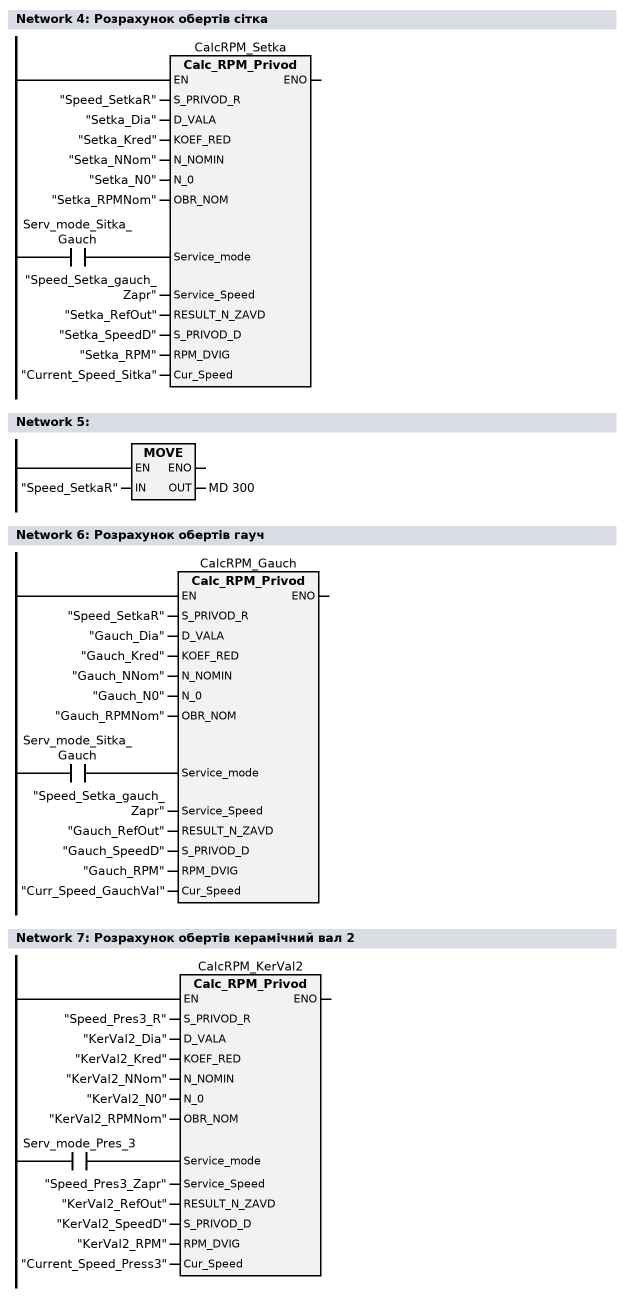
NETWORK
TITLE = Розрахунок обертів сітка
      A     "Serv_mode_Sitka_Gauch";
      =     L 0.0;
      BLD   103;
      CALL  "Calc_RPM_Privod" , "CalcRPM_Setka" (
           S_PRIVOD_R               := "Speed_SetkaR",
           D_VALA                   := "Setka_Dia",
           KOEF_RED                 := "Setka_Kred",
           N_NOMIN                  := "Setka_NNom",
           N_0                      := "Setka_N0",
           OBR_NOM                  := "Setka_RPMNom",
           Service_mode             := L 0.0,
           Service_Speed            := "Speed_Setka_gauch_Zapr",
           RESULT_N_ZAVD            := "Setka_RefOut",
           S_PRIVOD_D               := "Setka_SpeedD",
           RPM_DVIG                 := "Setka_RPM",
           Cur_Speed                := "Current_Speed_Sitka");
      NOP   0;
NETWORK
TITLE =
      L     "Speed_SetkaR";
      T     MD 300;
      NOP   0;
NETWORK
TITLE = Розрахунок обертів гауч
      A     "Serv_mode_Sitka_Gauch";
      =     L 0.0;
      BLD   103;
      CALL  "Calc_RPM_Privod" , "CalcRPM_Gauch" (
           S_PRIVOD_R               := "Speed_SetkaR",
           D_VALA                   := "Gauch_Dia",
           KOEF_RED                 := "Gauch_Kred",
           N_NOMIN                  := "Gauch_NNom",
           N_0                      := "Gauch_N0",
           OBR_NOM                  := "Gauch_RPMNom",
           Service_mode             := L 0.0,
           Service_Speed            := "Speed_Setka_gauch_Zapr",
           RESULT_N_ZAVD            := "Gauch_RefOut",
           S_PRIVOD_D               := "Gauch_SpeedD",
           RPM_DVIG                 := "Gauch_RPM",
           Cur_Speed                := "Curr_Speed_GauchVal");
      NOP   0;
NETWORK
TITLE = Розрахунок обертів керамічний вал 2
      A     "Serv_mode_Pres_3";
      =     L 0.0;
      BLD   103;
      CALL  "Calc_RPM_Privod" , "CalcRPM_KerVal2" (
           S_PRIVOD_R               := "Speed_Pres3_R",
           D_VALA                   := "KerVal2_Dia",
           KOEF_RED                 := "KerVal2_Kred",
           N_NOMIN                  := "KerVal2_NNom",
           N_0                      := "KerVal2_N0",
           OBR_NOM                  := "KerVal2_RPMNom",
           Service_mode             := L 0.0,
           Service_Speed            := "Speed_Pres3_Zapr",
           RESULT_N_ZAVD            := "KerVal2_RefOut",
           S_PRIVOD_D               := "KerVal2_SpeedD",
           RPM_DVIG                 := "KerVal2_RPM",
           Cur_Speed                := "Current_Speed_Press3");
      NOP   0;
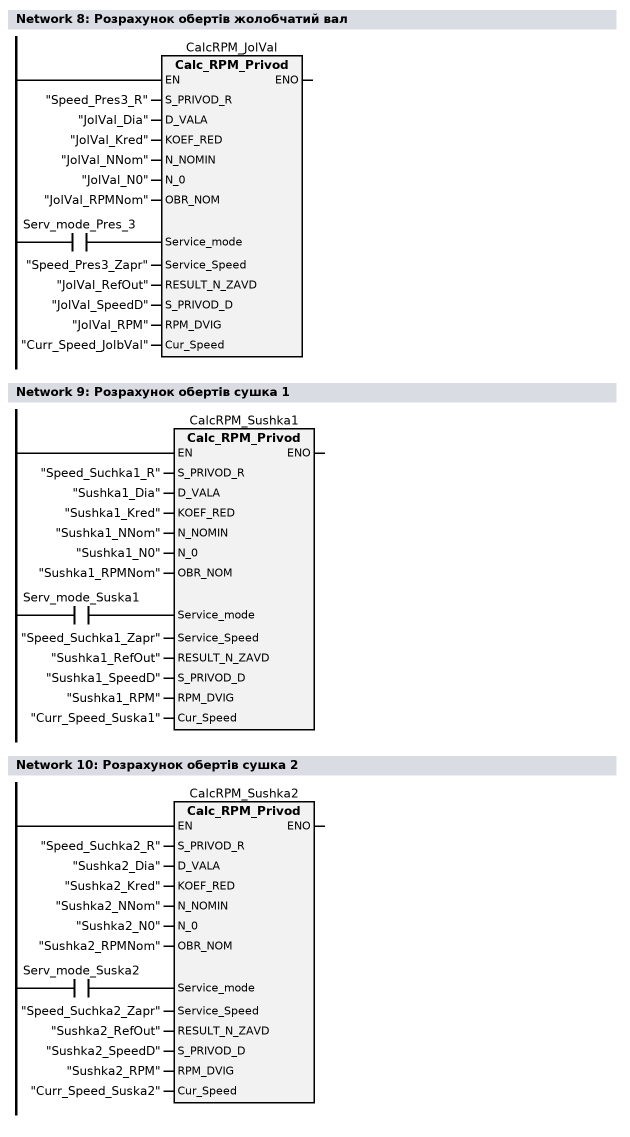
NETWORK
TITLE = Розрахунок обертів жолобчатий вал
      A     "Serv_mode_Pres_3";
      =     L 0.0;
      BLD   103;
      CALL  "Calc_RPM_Privod" , "CalcRPM_JolVal" (
           S_PRIVOD_R               := "Speed_Pres3_R",
           D_VALA                   := "JolVal_Dia",
           KOEF_RED                 := "JolVal_Kred",
           N_NOMIN                  := "JolVal_NNom",
           N_0                      := "JolVal_N0",
           OBR_NOM                  := "JolVal_RPMNom",
           Service_mode             := L 0.0,
           Service_Speed            := "Speed_Pres3_Zapr",
           RESULT_N_ZAVD            := "JolVal_RefOut",
           S_PRIVOD_D               := "JolVal_SpeedD",
           RPM_DVIG                 := "JolVal_RPM",
           Cur_Speed                := "Curr_Speed_JolbVal");
      NOP   0;
NETWORK
TITLE = Розрахунок обертів сушка 1
      A     "Serv_mode_Suska1";
      =     L 0.0;
      BLD   103;
      CALL  "Calc_RPM_Privod" , "CalcRPM_Sushka1" (
           S_PRIVOD_R               := "Speed_Suchka1_R",
           D_VALA                   := "Sushka1_Dia",
           KOEF_RED                 := "Sushka1_Kred",
           N_NOMIN                  := "Sushka1_NNom",
           N_0                      := "Sushka1_N0",
           OBR_NOM                  := "Sushka1_RPMNom",
           Service_mode             := L 0.0,
           Service_Speed            := "Speed_Suchka1_Zapr",
           RESULT_N_ZAVD            := "Sushka1_RefOut",
           S_PRIVOD_D               := "Sushka1_SpeedD",
           RPM_DVIG                 := "Sushka1_RPM",
           Cur_Speed                := "Curr_Speed_Suska1");
      NOP   0;
NETWORK
TITLE = Розрахунок обертів сушка 2
      A     "Serv_mode_Suska2";
      =     L 0.0;
      BLD   103;
      CALL  "Calc_RPM_Privod" , "CalcRPM_Sushka2" (
           S_PRIVOD_R               := "Speed_Suchka2_R",
           D_VALA                   := "Sushka2_Dia",
           KOEF_RED                 := "Sushka2_Kred",
           N_NOMIN                  := "Sushka2_NNom",
           N_0                      := "Sushka2_N0",
           OBR_NOM                  := "Sushka2_RPMNom",
           Service_mode             := L 0.0,
           Service_Speed            := "Speed_Suchka2_Zapr",
           RESULT_N_ZAVD            := "Sushka2_RefOut",
           S_PRIVOD_D               := "Sushka2_SpeedD",
           RPM_DVIG                 := "Sushka2_RPM",
           Cur_Speed                := "Curr_Speed_Suska2");
      NOP   0;
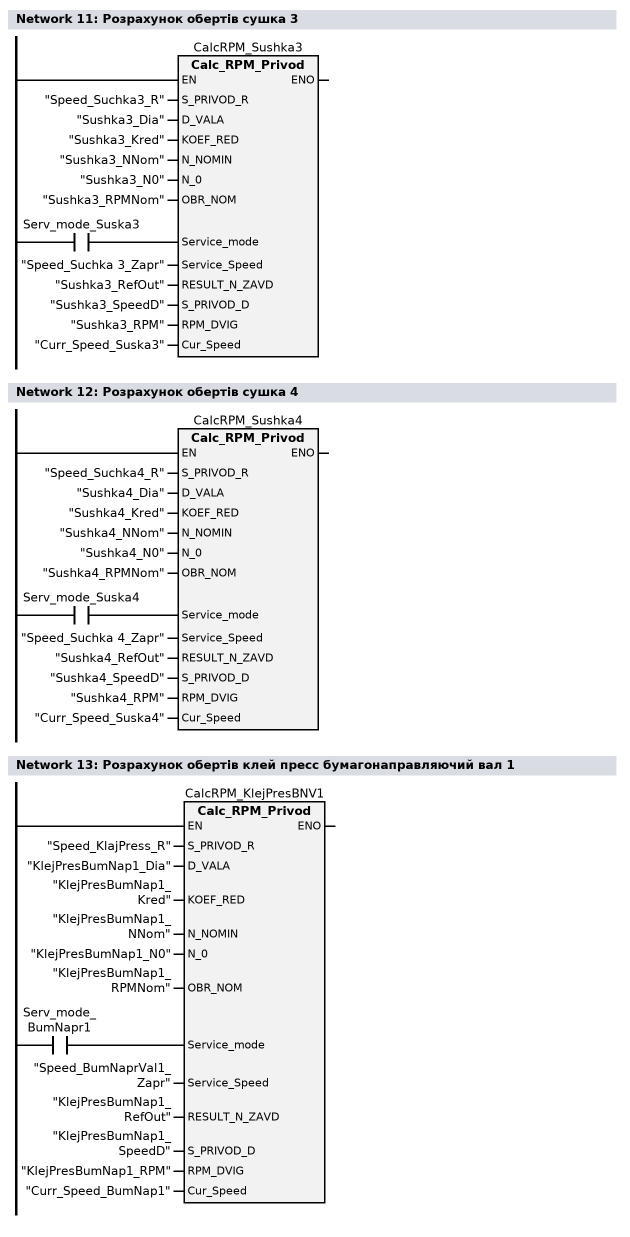
NETWORK
TITLE = Розрахунок обертів сушка 3
      A     "Serv_mode_Suska3";
      =     L 0.0;
      BLD   103;
      CALL  "Calc_RPM_Privod" , "CalcRPM_Sushka3" (
           S_PRIVOD_R               := "Speed_Suchka3_R",
           D_VALA                   := "Sushka3_Dia",
           KOEF_RED                 := "Sushka3_Kred",
           N_NOMIN                  := "Sushka3_NNom",
           N_0                      := "Sushka3_N0",
           OBR_NOM                  := "Sushka3_RPMNom",
           Service_mode             := L 0.0,
           Service_Speed            := "Speed_Suchka 3_Zapr",
           RESULT_N_ZAVD            := "Sushka3_RefOut",
           S_PRIVOD_D               := "Sushka3_SpeedD",
           RPM_DVIG                 := "Sushka3_RPM",
           Cur_Speed                := "Curr_Speed_Suska3");
      NOP   0;
NETWORK
TITLE = Розрахунок обертів сушка 4
      A     "Serv_mode_Suska4";
      =     L 0.0;
      BLD   103;
      CALL  "Calc_RPM_Privod" , "CalcRPM_Sushka4" (
           S_PRIVOD_R               := "Speed_Suchka4_R",
           D_VALA                   := "Sushka4_Dia",
           KOEF_RED                 := "Sushka4_Kred",
           N_NOMIN                  := "Sushka4_NNom",
           N_0                      := "Sushka4_N0",
           OBR_NOM                  := "Sushka4_RPMNom",
           Service_mode             := L 0.0,
           Service_Speed            := "Speed_Suchka 4_Zapr",
           RESULT_N_ZAVD            := "Sushka4_RefOut",
           S_PRIVOD_D               := "Sushka4_SpeedD",
           RPM_DVIG                 := "Sushka4_RPM",
           Cur_Speed                := "Curr_Speed_Suska4");
      NOP   0;
NETWORK
TITLE = Розрахунок обертів клей пресс бумагонаправляючий вал 1
      A     "Serv_mode_BumNapr1";
      =     L 0.0;
      BLD   103;
      CALL  "Calc_RPM_Privod" , "CalcRPM_KlejPresBNV1" (
           S_PRIVOD_R               := "Speed_KlajPress_R",
           D_VALA                   := "KlejPresBumNap1_Dia",
           KOEF_RED                 := "KlejPresBumNap1_Kred",
           N_NOMIN                  := "KlejPresBumNap1_NNom",
           N_0                      := "KlejPresBumNap1_N0",
           OBR_NOM                  := "KlejPresBumNap1_RPMNom",
           Service_mode             := L 0.0,
           Service_Speed            := "Speed_BumNaprVal1_Zapr",
           RESULT_N_ZAVD            := "KlejPresBumNap1_RefOut",
           S_PRIVOD_D               := "KlejPresBumNap1_SpeedD",
           RPM_DVIG                 := "KlejPresBumNap1_RPM",
           Cur_Speed                := "Curr_Speed_BumNap1");
      NOP   0;
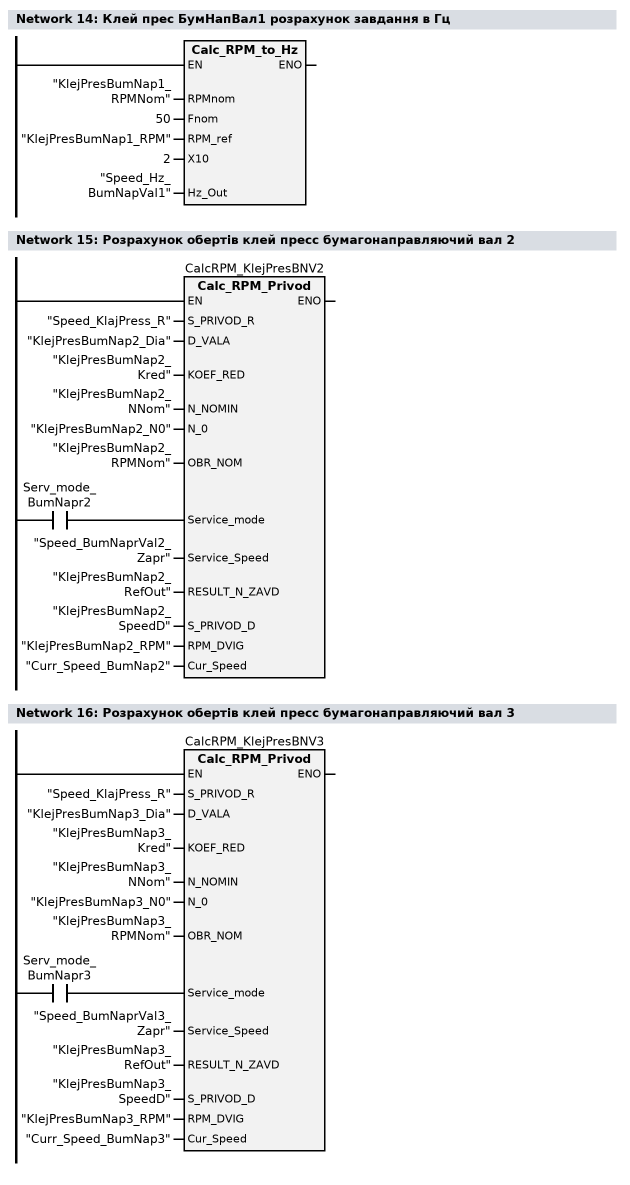
NETWORK
TITLE = Клей прес БумНапВал1 розрахунок завдання в Гц
      CALL  "Calc_RPM_to_Hz" (
           RPMnom                   := "KlejPresBumNap1_RPMNom",
           Fnom                     := 50,
           RPM_ref                  := "KlejPresBumNap1_RPM",
           X10                      := 2,
           Hz_Out                   := "Speed_Hz_BumNapVal1");
      NOP   0;
NETWORK
TITLE = Розрахунок обертів клей пресс бумагонаправляючий вал 2
      A     "Serv_mode_BumNapr2";
      =     L 0.0;
      BLD   103;
      CALL  "Calc_RPM_Privod" , "CalcRPM_KlejPresBNV2" (
           S_PRIVOD_R               := "Speed_KlajPress_R",
           D_VALA                   := "KlejPresBumNap2_Dia",
           KOEF_RED                 := "KlejPresBumNap2_Kred",
           N_NOMIN                  := "KlejPresBumNap2_NNom",
           N_0                      := "KlejPresBumNap2_N0",
           OBR_NOM                  := "KlejPresBumNap2_RPMNom",
           Service_mode             := L 0.0,
           Service_Speed            := "Speed_BumNaprVal2_Zapr",
           RESULT_N_ZAVD            := "KlejPresBumNap2_RefOut",
           S_PRIVOD_D               := "KlejPresBumNap2_SpeedD",
           RPM_DVIG                 := "KlejPresBumNap2_RPM",
           Cur_Speed                := "Curr_Speed_BumNap2");
      NOP   0;
NETWORK
TITLE = Розрахунок обертів клей пресс бумагонаправляючий вал 3
      A     "Serv_mode_BumNapr3";
      =     L 0.0;
      BLD   103;
      CALL  "Calc_RPM_Privod" , "CalcRPM_KlejPresBNV3" (
           S_PRIVOD_R               := "Speed_KlajPress_R",
           D_VALA                   := "KlejPresBumNap3_Dia",
           KOEF_RED                 := "KlejPresBumNap3_Kred",
           N_NOMIN                  := "KlejPresBumNap3_NNom",
           N_0                      := "KlejPresBumNap3_N0",
           OBR_NOM                  := "KlejPresBumNap3_RPMNom",
           Service_mode             := L 0.0,
           Service_Speed            := "Speed_BumNaprVal3_Zapr",
           RESULT_N_ZAVD            := "KlejPresBumNap3_RefOut",
           S_PRIVOD_D               := "KlejPresBumNap3_SpeedD",
           RPM_DVIG                 := "KlejPresBumNap3_RPM",
           Cur_Speed                := "Curr_Speed_BumNap3");
      NOP   0;
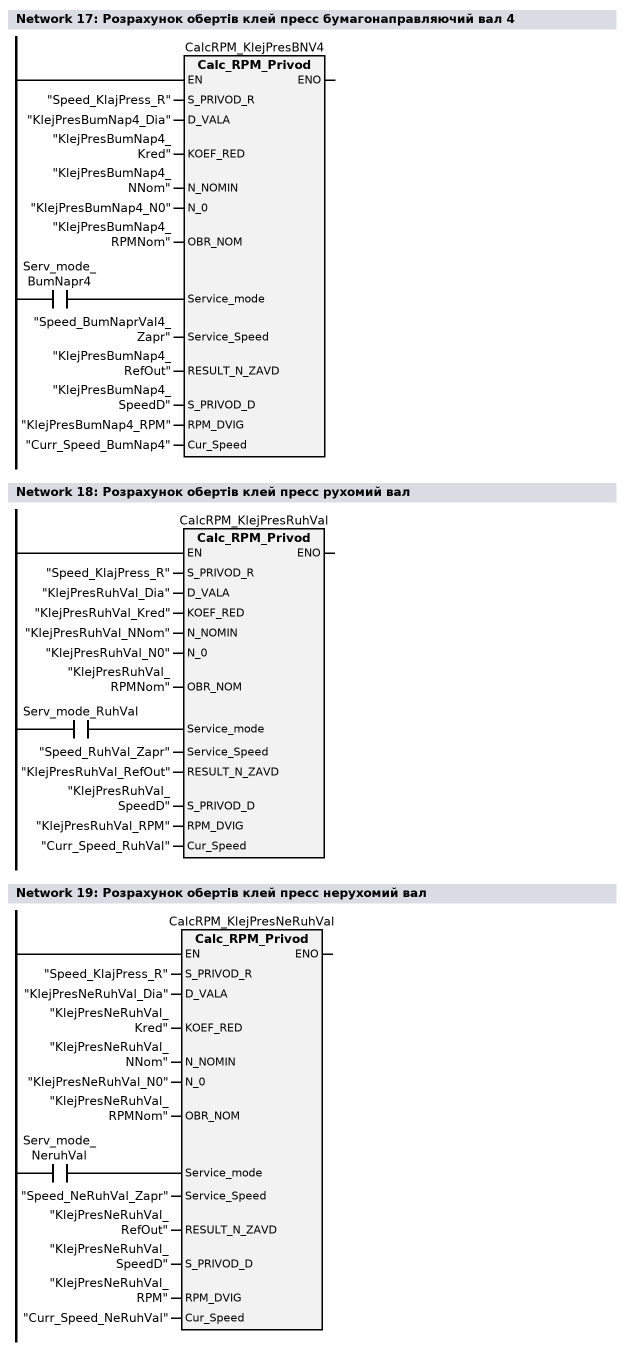
NETWORK
TITLE = Розрахунок обертів клей пресс бумагонаправляючий вал 4
      A     "Serv_mode_BumNapr4";
      =     L 0.0;
      BLD   103;
      CALL  "Calc_RPM_Privod" , "CalcRPM_KlejPresBNV4" (
           S_PRIVOD_R               := "Speed_KlajPress_R",
           D_VALA                   := "KlejPresBumNap4_Dia",
           KOEF_RED                 := "KlejPresBumNap4_Kred",
           N_NOMIN                  := "KlejPresBumNap4_NNom",
           N_0                      := "KlejPresBumNap4_N0",
           OBR_NOM                  := "KlejPresBumNap4_RPMNom",
           Service_mode             := L 0.0,
           Service_Speed            := "Speed_BumNaprVal4_Zapr",
           RESULT_N_ZAVD            := "KlejPresBumNap4_RefOut",
           S_PRIVOD_D               := "KlejPresBumNap4_SpeedD",
           RPM_DVIG                 := "KlejPresBumNap4_RPM",
           Cur_Speed                := "Curr_Speed_BumNap4");
      NOP   0;
NETWORK
TITLE = Розрахунок обертів клей пресс рухомий вал
      A     "Serv_mode_RuhVal";
      =     L 0.0;
      BLD   103;
      CALL  "Calc_RPM_Privod" , "CalcRPM_KlejPresRuhVal" (
           S_PRIVOD_R               := "Speed_KlajPress_R",
           D_VALA                   := "KlejPresRuhVal_Dia",
           KOEF_RED                 := "KlejPresRuhVal_Kred",
           N_NOMIN                  := "KlejPresRuhVal_NNom",
           N_0                      := "KlejPresRuhVal_N0",
           OBR_NOM                  := "KlejPresRuhVal_RPMNom",
           Service_mode             := L 0.0,
           Service_Speed            := "Speed_RuhVal_Zapr",
           RESULT_N_ZAVD            := "KlejPresRuhVal_RefOut",
           S_PRIVOD_D               := "KlejPresRuhVal_SpeedD",
           RPM_DVIG                 := "KlejPresRuhVal_RPM",
           Cur_Speed                := "Curr_Speed_RuhVal");
      NOP   0;
NETWORK
TITLE = Розрахунок обертів клей пресс нерухомий вал
      A     "Serv_mode_NeruhVal";
      =     L 0.0;
      BLD   103;
      CALL  "Calc_RPM_Privod" , "CalcRPM_KlejPresNeRuhVal" (
           S_PRIVOD_R               := "Speed_KlajPress_R",
           D_VALA                   := "KlejPresNeRuhVal_Dia",
           KOEF_RED                 := "KlejPresNeRuhVal_Kred",
           N_NOMIN                  := "KlejPresNeRuhVal_NNom",
           N_0                      := "KlejPresNeRuhVal_N0",
           OBR_NOM                  := "KlejPresNeRuhVal_RPMNom",
           Service_mode             := L 0.0,
           Service_Speed            := "Speed_NeRuhVal_Zapr",
           RESULT_N_ZAVD            := "KlejPresNeRuhVal_RefOut",
           S_PRIVOD_D               := "KlejPresNeRuhVal_SpeedD",
           RPM_DVIG                 := "KlejPresNeRuhVal_RPM",
           Cur_Speed                := "Curr_Speed_NeRuhVal");
      NOP   0;
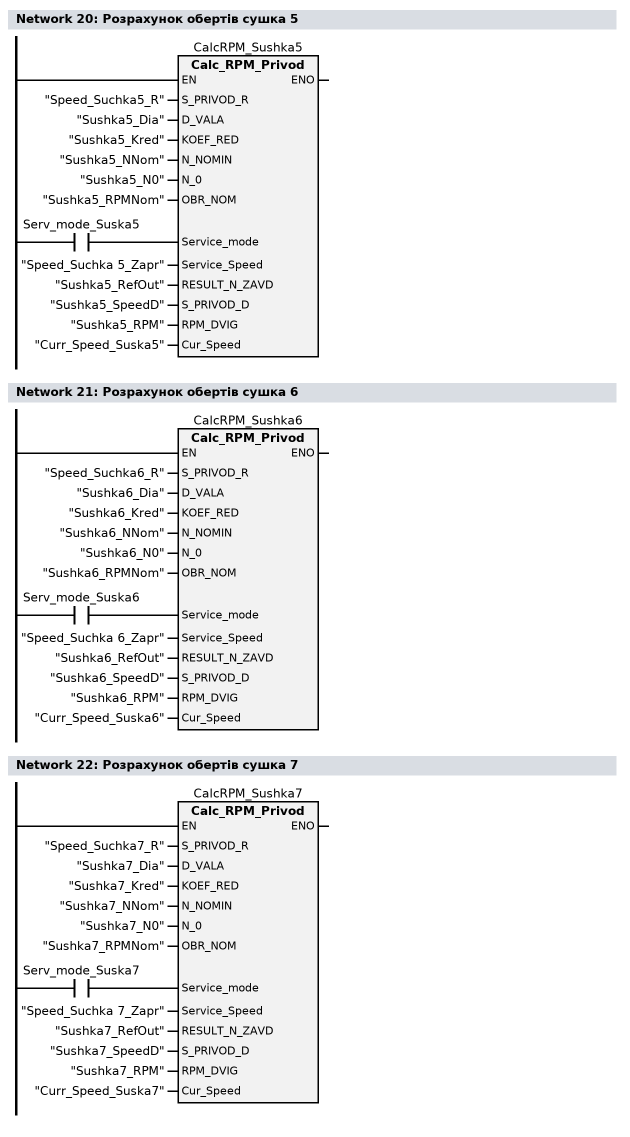
NETWORK
TITLE = Розрахунок обертів сушка 5
      A     "Serv_mode_Suska5";
      =     L 0.0;
      BLD   103;
      CALL  "Calc_RPM_Privod" , "CalcRPM_Sushka5" (
           S_PRIVOD_R               := "Speed_Suchka5_R",
           D_VALA                   := "Sushka5_Dia",
           KOEF_RED                 := "Sushka5_Kred",
           N_NOMIN                  := "Sushka5_NNom",
           N_0                      := "Sushka5_N0",
           OBR_NOM                  := "Sushka5_RPMNom",
           Service_mode             := L 0.0,
           Service_Speed            := "Speed_Suchka 5_Zapr",
           RESULT_N_ZAVD            := "Sushka5_RefOut",
           S_PRIVOD_D               := "Sushka5_SpeedD",
           RPM_DVIG                 := "Sushka5_RPM",
           Cur_Speed                := "Curr_Speed_Suska5");
      NOP   0;
NETWORK
TITLE = Розрахунок обертів сушка 6
      A     "Serv_mode_Suska6";
      =     L 0.0;
      BLD   103;
      CALL  "Calc_RPM_Privod" , "CalcRPM_Sushka6" (
           S_PRIVOD_R               := "Speed_Suchka6_R",
           D_VALA                   := "Sushka6_Dia",
           KOEF_RED                 := "Sushka6_Kred",
           N_NOMIN                  := "Sushka6_NNom",
           N_0                      := "Sushka6_N0",
           OBR_NOM                  := "Sushka6_RPMNom",
           Service_mode             := L 0.0,
           Service_Speed            := "Speed_Suchka 6_Zapr",
           RESULT_N_ZAVD            := "Sushka6_RefOut",
           S_PRIVOD_D               := "Sushka6_SpeedD",
           RPM_DVIG                 := "Sushka6_RPM",
           Cur_Speed                := "Curr_Speed_Suska6");
      NOP   0;
NETWORK
TITLE = Розрахунок обертів сушка 7
      A     "Serv_mode_Suska7";
      =     L 0.0;
      BLD   103;
      CALL  "Calc_RPM_Privod" , "CalcRPM_Sushka7" (
           S_PRIVOD_R               := "Speed_Suchka7_R",
           D_VALA                   := "Sushka7_Dia",
           KOEF_RED                 := "Sushka7_Kred",
           N_NOMIN                  := "Sushka7_NNom",
           N_0                      := "Sushka7_N0",
           OBR_NOM                  := "Sushka7_RPMNom",
           Service_mode             := L 0.0,
           Service_Speed            := "Speed_Suchka 7_Zapr",
           RESULT_N_ZAVD            := "Sushka7_RefOut",
           S_PRIVOD_D               := "Sushka7_SpeedD",
           RPM_DVIG                 := "Sushka7_RPM",
           Cur_Speed                := "Curr_Speed_Suska7");
      NOP   0;
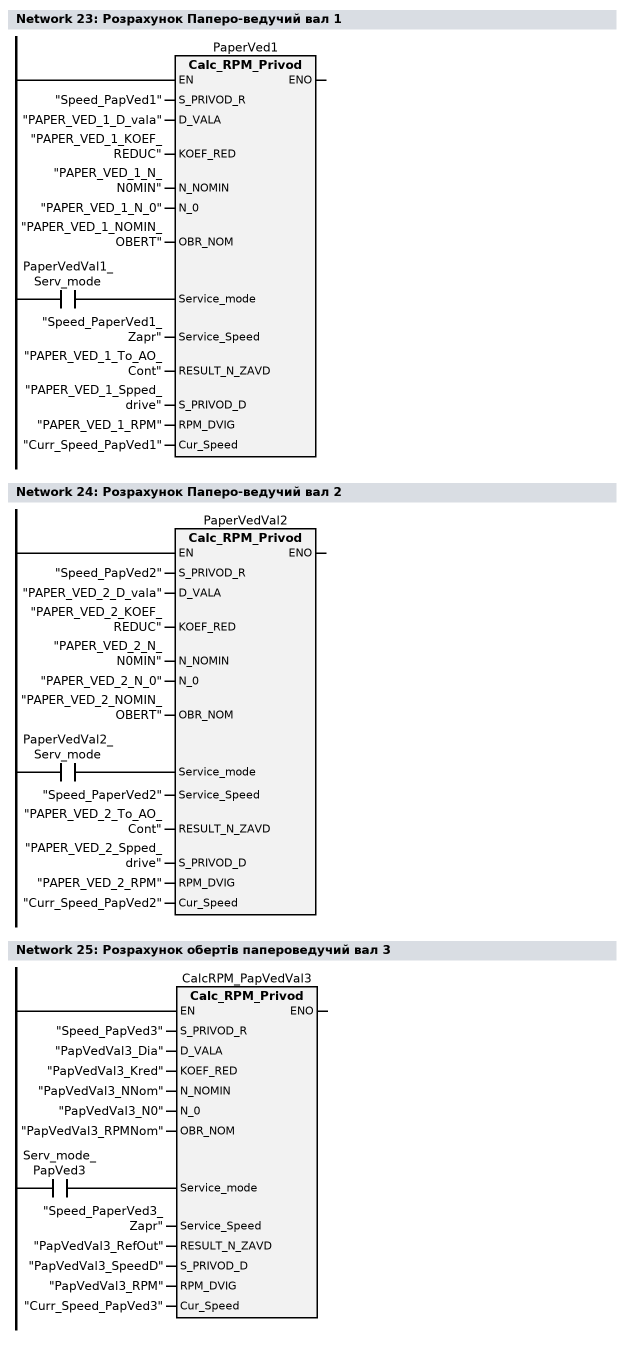
NETWORK
TITLE = Розрахунок Паперо-ведучий вал 1
//********************************************
//
      A     "PaperVedVal1_Serv_mode";
      =     L 0.0;
      BLD   103;
      CALL  "Calc_RPM_Privod" , "PaperVed1" (
           S_PRIVOD_R               := "Speed_PapVed1",
           D_VALA                   := "PAPER_VED_1_D_vala",
           KOEF_RED                 := "PAPER_VED_1_KOEF_REDUC",
           N_NOMIN                  := "PAPER_VED_1_N_N0MIN",
           N_0                      := "PAPER_VED_1_N_0",
           OBR_NOM                  := "PAPER_VED_1_NOMIN_OBERT",
           Service_mode             := L 0.0,
           Service_Speed            := "Speed_PaperVed1_Zapr",
           RESULT_N_ZAVD            := "PAPER_VED_1_To_AO_Cont",
           S_PRIVOD_D               := "PAPER_VED_1_Spped_drive",
           RPM_DVIG                 := "PAPER_VED_1_RPM",
           Cur_Speed                := "Curr_Speed_PapVed1");
      NOP   0;
NETWORK
TITLE = Розрахунок Паперо-ведучий вал 2
//*********************************************
//
      A     "PaperVedVal2_Serv_mode";
      =     L 0.0;
      BLD   103;
      CALL  "Calc_RPM_Privod" , "PaperVedVal2" (
           S_PRIVOD_R               := "Speed_PapVed2",
           D_VALA                   := "PAPER_VED_2_D_vala",
           KOEF_RED                 := "PAPER_VED_2_KOEF_REDUC",
           N_NOMIN                  := "PAPER_VED_2_N_N0MIN",
           N_0                      := "PAPER_VED_2_N_0",
           OBR_NOM                  := "PAPER_VED_2_NOMIN_OBERT",
           Service_mode             := L 0.0,
           Service_Speed            := "Speed_PaperVed2",
           RESULT_N_ZAVD            := "PAPER_VED_2_To_AO_Cont",
           S_PRIVOD_D               := "PAPER_VED_2_Spped_drive",
           RPM_DVIG                 := "PAPER_VED_2_RPM",
           Cur_Speed                := "Curr_Speed_PapVed2");
      NOP   0;
NETWORK
TITLE = Розрахунок обертів папероведучий вал 3
//****************************************************
//
      A     "Serv_mode_PapVed3";
      =     L 0.0;
      BLD   103;
      CALL  "Calc_RPM_Privod" , "CalcRPM_PapVedVal3" (
           S_PRIVOD_R               := "Speed_PapVed3",
           D_VALA                   := "PapVedVal3_Dia",
           KOEF_RED                 := "PapVedVal3_Kred",
           N_NOMIN                  := "PapVedVal3_NNom",
           N_0                      := "PapVedVal3_N0",
           OBR_NOM                  := "PapVedVal3_RPMNom",
           Service_mode             := L 0.0,
           Service_Speed            := "Speed_PaperVed3_Zapr",
           RESULT_N_ZAVD            := "PapVedVal3_RefOut",
           S_PRIVOD_D               := "PapVedVal3_SpeedD",
           RPM_DVIG                 := "PapVedVal3_RPM",
           Cur_Speed                := "Curr_Speed_PapVed3");
      NOP   0;
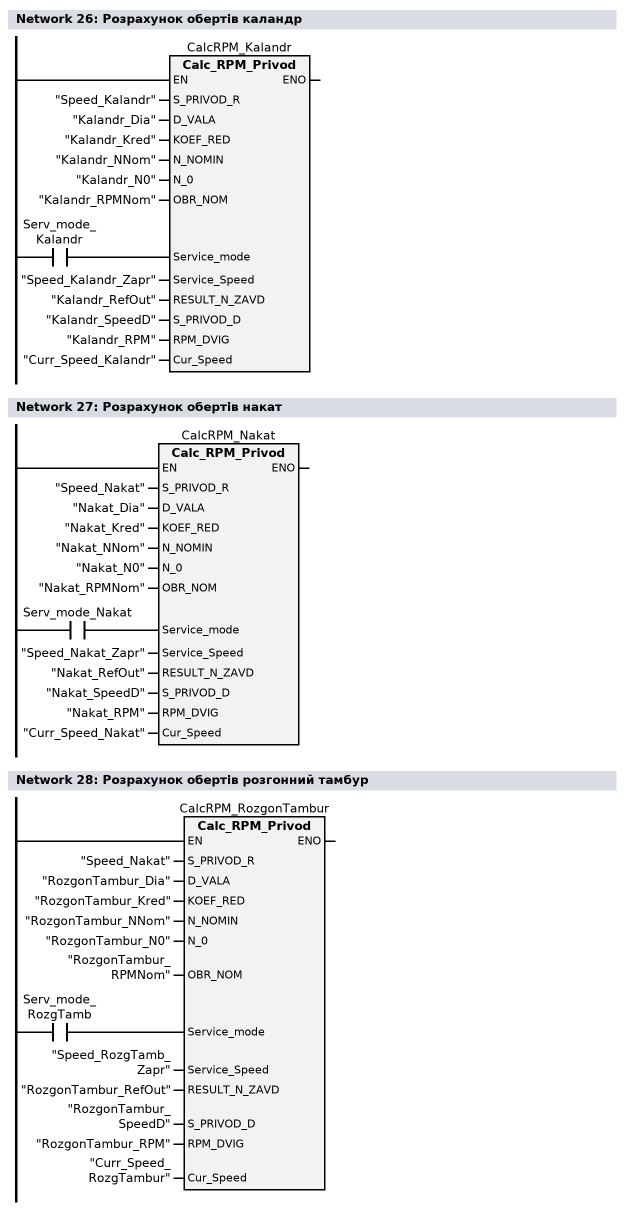
NETWORK
TITLE = Розрахунок обертів каландр
      A     "Serv_mode_Kalandr";
      =     L 0.0;
      BLD   103;
      CALL  "Calc_RPM_Privod" , "CalcRPM_Kalandr" (
           S_PRIVOD_R               := "Speed_Kalandr",
           D_VALA                   := "Kalandr_Dia",
           KOEF_RED                 := "Kalandr_Kred",
           N_NOMIN                  := "Kalandr_NNom",
           N_0                      := "Kalandr_N0",
           OBR_NOM                  := "Kalandr_RPMNom",
           Service_mode             := L 0.0,
           Service_Speed            := "Speed_Kalandr_Zapr",
           RESULT_N_ZAVD            := "Kalandr_RefOut",
           S_PRIVOD_D               := "Kalandr_SpeedD",
           RPM_DVIG                 := "Kalandr_RPM",
           Cur_Speed                := "Curr_Speed_Kalandr");
      NOP   0;
NETWORK
TITLE = Розрахунок обертів накат
      A     "Serv_mode_Nakat";
      =     L 0.0;
      BLD   103;
      CALL  "Calc_RPM_Privod" , "CalcRPM_Nakat" (
           S_PRIVOD_R               := "Speed_Nakat",
           D_VALA                   := "Nakat_Dia",
           KOEF_RED                 := "Nakat_Kred",
           N_NOMIN                  := "Nakat_NNom",
           N_0                      := "Nakat_N0",
           OBR_NOM                  := "Nakat_RPMNom",
           Service_mode             := L 0.0,
           Service_Speed            := "Speed_Nakat_Zapr",
           RESULT_N_ZAVD            := "Nakat_RefOut",
           S_PRIVOD_D               := "Nakat_SpeedD",
           RPM_DVIG                 := "Nakat_RPM",
           Cur_Speed                := "Curr_Speed_Nakat");
      NOP   0;
NETWORK
TITLE = Розрахунок обертів розгонний тамбур
      A     "Serv_mode_RozgTamb";
      =     L 0.0;
      BLD   103;
      CALL  "Calc_RPM_Privod" , "CalcRPM_RozgonTambur" (
           S_PRIVOD_R               := "Speed_Nakat",
           D_VALA                   := "RozgonTambur_Dia",
           KOEF_RED                 := "RozgonTambur_Kred",
           N_NOMIN                  := "RozgonTambur_NNom",
           N_0                      := "RozgonTambur_N0",
           OBR_NOM                  := "RozgonTambur_RPMNom",
           Service_mode             := L 0.0,
           Service_Speed            := "Speed_RozgTamb_Zapr",
           RESULT_N_ZAVD            := "RozgonTambur_RefOut",
           S_PRIVOD_D               := "RozgonTambur_SpeedD",
           RPM_DVIG                 := "RozgonTambur_RPM",
           Cur_Speed                := "Curr_Speed_RozgTambur");
      NOP   0;
END_FUNCTION

FUNCTION "Speed_Intens" : VOID	// FC 12
VERSION : 0.1
VAR_TEMP
  Speed_1R : REAL ;
END_VAR
BEGIN
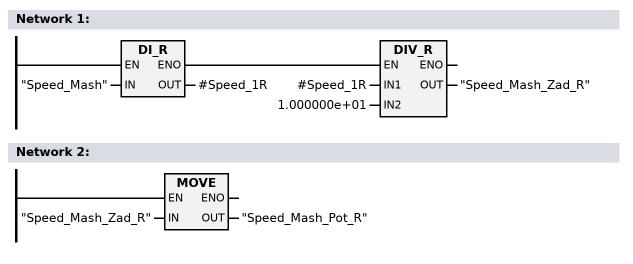
NETWORK
TITLE =
      A(;
      L     "Speed_Mash";
      DTR;
      T     #Speed_1R;
      SET;
      SAVE;
      CLR;
      A     BR;
      );
      JNB   _001;
      L     #Speed_1R;
      L     1.000000e+01;
      /R;
      T     "Speed_Mash_Zad_R";
_001: NOP   0;
NETWORK
TITLE =
      L     "Speed_Mash_Zad_R";
      T     "Speed_Mash_Pot_R";
      NOP   0;
END_FUNCTION

FUNCTION "Calc_RPM_to_Hz" : VOID	// FC 14
VERSION : 0.1
VAR_INPUT
  RPMnom : DINT ;
  Fnom : INT ;
  RPM_ref : DINT ;
  X10 : INT ;
END_VAR
VAR_OUTPUT
  Hz_Out : WORD ;
END_VAR
VAR_TEMP
  Fn_R : REAL ;
  Rn_R : REAL ;
  Rz_R : REAL ;
  Fnom_DI : DINT ;
  TEMP0 : REAL ;
  Fref_R : REAL ;
  TEMP10 : REAL ;
  TEMP1 : REAL ;
  Hz_Out_DI : DINT ;
END_VAR
BEGIN
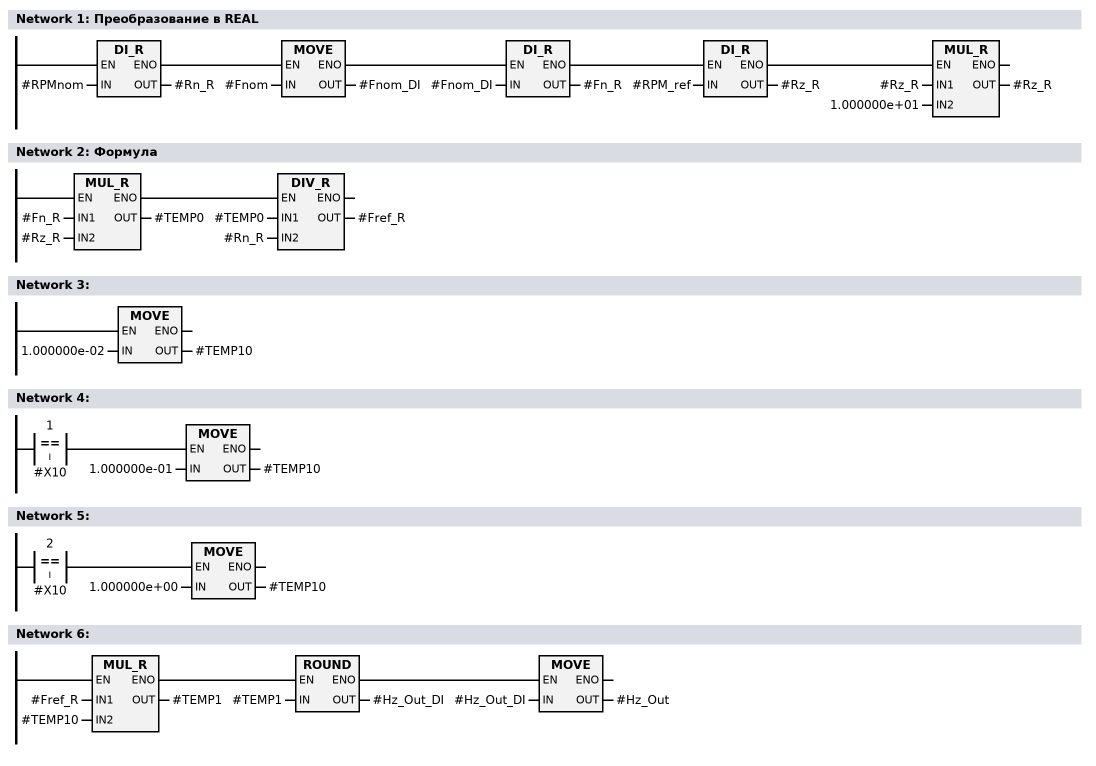
NETWORK
TITLE = Преобразование в REAL
      A(;
      A(;
      A(;
      A(;
      L     #RPMnom;
      DTR;
      T     #Rn_R;
      SET;
      SAVE;
      CLR;
      A     BR;
      );
      JNB   _001;
      L     #Fnom;
      T     #Fnom_DI;
      SET;
      SAVE;
      CLR;
_001: A     BR;
      );
      JNB   _002;
      L     #Fnom_DI;
      DTR;
      T     #Fn_R;
      SET;
      SAVE;
      CLR;
_002: A     BR;
      );
      JNB   _003;
      L     #RPM_ref;
      DTR;
      T     #Rz_R;
      SET;
      SAVE;
      CLR;
_003: A     BR;
      );
      JNB   _004;
      L     #Rz_R;
      L     1.000000e+01;
      *R;
      T     #Rz_R;
_004: NOP   0;
NETWORK
TITLE = Формула
      A(;
      L     #Fn_R;
      L     #Rz_R;
      *R;
      T     #TEMP0;
      AN    OV;
      SAVE;
      CLR;
      A     BR;
      );
      JNB   _005;
      L     #TEMP0;
      L     #Rn_R;
      /R;
      T     #Fref_R;
_005: NOP   0;
NETWORK
TITLE =
      L     1.000000e-02;
      T     #TEMP10;
      NOP   0;
NETWORK
TITLE =
      A(;
      L     1;
      L     #X10;
      ==I;
      );
      JNB   _006;
      L     1.000000e-01;
      T     #TEMP10;
_006: NOP   0;
NETWORK
TITLE =
      A(;
      L     2;
      L     #X10;
      ==I;
      );
      JNB   _007;
      L     1.000000e+00;
      T     #TEMP10;
_007: NOP   0;
NETWORK
TITLE =
      A(;
      A(;
      L     #Fref_R;
      L     #TEMP10;
      *R;
      T     #TEMP1;
      AN    OV;
      SAVE;
      CLR;
      A     BR;
      );
      JNB   _008;
      L     #TEMP1;
      RND;
      T     #Hz_Out_DI;
      AN    OV;
      SAVE;
      CLR;
_008: A     BR;
      );
      JNB   _009;
      L     #Hz_Out_DI;
      T     #Hz_Out;
_009: NOP   0;
END_FUNCTION

FUNCTION "Check_AlarmPPS" : VOID	// FC 30
VERSION : 0.1
VAR_INPUT
  Key_FU : BOOL ;
  Key_DozvilRun : BOOL ;
  Blokuvannja : BOOL ;
  AlarmPryvid : BOOL ;
  Warnunug_T : BOOL ;
  Alarm_T : BOOL ;
END_VAR
VAR_OUTPUT
  Cod_Err : WORD ;
  Privod_OK : BOOL ;
END_VAR
VAR_TEMP
  TEMP : BOOL ;
END_VAR
BEGIN
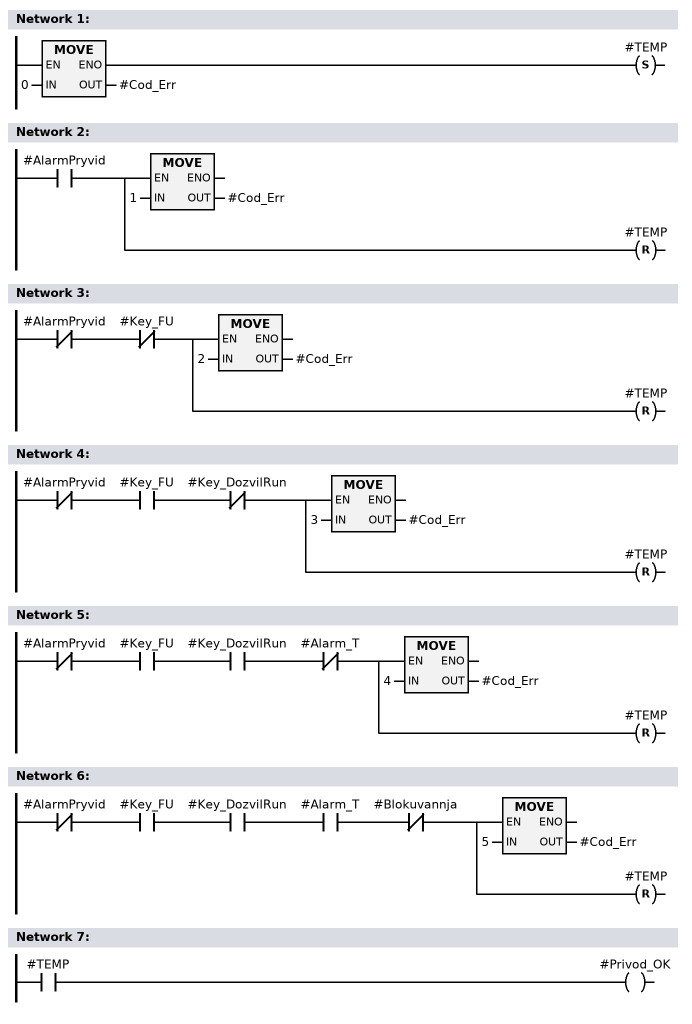
NETWORK
TITLE =
      L     0;
      T     #Cod_Err;
      SET;
      SAVE;
      CLR;
      A     BR;
      S     #TEMP;
NETWORK
TITLE =
      A     #AlarmPryvid;
      =     L 1.0;
      A     L 1.0;
      JNB   _001;
      L     1;
      T     #Cod_Err;
_001: NOP   0;
      A     L 1.0;
      BLD   102;
      R     #TEMP;
NETWORK
TITLE =
      AN    #AlarmPryvid;
      AN    #Key_FU;
      =     L 1.0;
      A     L 1.0;
      JNB   _002;
      L     2;
      T     #Cod_Err;
_002: NOP   0;
      A     L 1.0;
      BLD   102;
      R     #TEMP;
NETWORK
TITLE =
      AN    #AlarmPryvid;
      A     #Key_FU;
      AN    #Key_DozvilRun;
      =     L 1.0;
      A     L 1.0;
      JNB   _003;
      L     3;
      T     #Cod_Err;
_003: NOP   0;
      A     L 1.0;
      BLD   102;
      R     #TEMP;
NETWORK
TITLE =
      AN    #AlarmPryvid;
      A     #Key_FU;
      A     #Key_DozvilRun;
      AN    #Alarm_T;
      =     L 1.0;
      A     L 1.0;
      JNB   _004;
      L     4;
      T     #Cod_Err;
_004: NOP   0;
      A     L 1.0;
      BLD   102;
      R     #TEMP;
NETWORK
TITLE =
      AN    #AlarmPryvid;
      A     #Key_FU;
      A     #Key_DozvilRun;
      A     #Alarm_T;
      AN    #Blokuvannja;
      =     L 1.0;
      A     L 1.0;
      JNB   _005;
      L     5;
      T     #Cod_Err;
_005: NOP   0;
      A     L 1.0;
      BLD   102;
      R     #TEMP;
NETWORK
TITLE =
      A     #TEMP;
      =     #Privod_OK;
END_FUNCTION

// FC 216: know-how protected block, not included

DATA_BLOCK DB 60
VERSION : 0.0
"SEND"
BEGIN
END_DATA_BLOCK

DATA_BLOCK DB 61
VERSION : 0.0
"RECEIVE"
BEGIN
END_DATA_BLOCK

DATA_BLOCK "RS485_chenal1"	// DB 71
AUTHOR : VIPA
FAMILY : MODBUS
VERSION : 0.0
"RTU_MB_MASTER"
BEGIN
END_DATA_BLOCK

DATA_BLOCK "RS485_chanel2"	// DB 72
AUTHOR : VIPA
FAMILY : MODBUS
VERSION : 0.1
"RTU_MB_MASTER"
BEGIN
END_DATA_BLOCK

DATA_BLOCK "RS485_chanel3"	// DB 73
AUTHOR : VIPA
FAMILY : MODBUS
VERSION : 0.0
"RTU_MB_MASTER"
BEGIN
END_DATA_BLOCK

DATA_BLOCK "RS485_chanel4"	// DB 74
AUTHOR : VIPA
FAMILY : MODBUS
VERSION : 0.0
"RTU_MB_MASTER"
BEGIN
END_DATA_BLOCK

DATA_BLOCK "KerVal1"	// DB 101
VERSION : 0.1
"Calc_RPM_Privod"
BEGIN
END_DATA_BLOCK

DATA_BLOCK "ValGluchPerf"	// DB 102
VERSION : 0.0
"Calc_RPM_Privod"
BEGIN
END_DATA_BLOCK

DATA_BLOCK "VidsmokVal"	// DB 103
VERSION : 0.0
"Calc_RPM_Privod"
BEGIN
END_DATA_BLOCK

DATA_BLOCK "CalcRPM_Setka"	// DB 104
VERSION : 0.0
"Calc_RPM_Privod"
BEGIN
END_DATA_BLOCK

DATA_BLOCK "CalcRPM_Gauch"	// DB 105
VERSION : 0.0
"Calc_RPM_Privod"
BEGIN
END_DATA_BLOCK

DATA_BLOCK "CalcRPM_KerVal2"	// DB 106
VERSION : 0.0
"Calc_RPM_Privod"
BEGIN
END_DATA_BLOCK

DATA_BLOCK "CalcRPM_JolVal"	// DB 107
VERSION : 0.0
"Calc_RPM_Privod"
BEGIN
END_DATA_BLOCK

DATA_BLOCK "CalcRPM_Sushka1"	// DB 108
VERSION : 0.0
"Calc_RPM_Privod"
BEGIN
END_DATA_BLOCK

DATA_BLOCK "CalcRPM_Sushka2"	// DB 109
VERSION : 0.0
"Calc_RPM_Privod"
BEGIN
END_DATA_BLOCK

DATA_BLOCK "CalcRPM_Sushka3"	// DB 110
VERSION : 0.0
"Calc_RPM_Privod"
BEGIN
END_DATA_BLOCK

DATA_BLOCK "CalcRPM_Sushka4"	// DB 111
VERSION : 0.0
"Calc_RPM_Privod"
BEGIN
END_DATA_BLOCK

DATA_BLOCK "CalcRPM_KlejPresBNV1"	// DB 112
VERSION : 0.0
"Calc_RPM_Privod"
BEGIN
END_DATA_BLOCK

DATA_BLOCK "CalcRPM_KlejPresBNV2"	// DB 113
VERSION : 0.0
"Calc_RPM_Privod"
BEGIN
END_DATA_BLOCK

DATA_BLOCK "CalcRPM_KlejPresBNV3"	// DB 114
VERSION : 0.0
"Calc_RPM_Privod"
BEGIN
END_DATA_BLOCK

DATA_BLOCK "CalcRPM_KlejPresBNV4"	// DB 115
VERSION : 0.0
"Calc_RPM_Privod"
BEGIN
END_DATA_BLOCK

DATA_BLOCK "CalcRPM_KlejPresRuhVal"	// DB 116
VERSION : 0.0
"Calc_RPM_Privod"
BEGIN
END_DATA_BLOCK

DATA_BLOCK "CalcRPM_KlejPresNeRuhVal"	// DB 117
VERSION : 0.0
"Calc_RPM_Privod"
BEGIN
END_DATA_BLOCK

DATA_BLOCK "CalcRPM_Sushka5"	// DB 118
VERSION : 0.0
"Calc_RPM_Privod"
BEGIN
END_DATA_BLOCK

DATA_BLOCK "CalcRPM_Sushka6"	// DB 119
VERSION : 0.0
"Calc_RPM_Privod"
BEGIN
END_DATA_BLOCK

DATA_BLOCK "CalcRPM_Sushka7"	// DB 120
VERSION : 0.0
"Calc_RPM_Privod"
BEGIN
END_DATA_BLOCK

DATA_BLOCK "CalcRPM_Kalandr"	// DB 121
VERSION : 0.0
"Calc_RPM_Privod"
BEGIN
END_DATA_BLOCK

DATA_BLOCK "CalcRPM_Nakat"	// DB 122
VERSION : 0.0
"Calc_RPM_Privod"
BEGIN
END_DATA_BLOCK

DATA_BLOCK "PaperVed1"	// DB 123
VERSION : 0.0
"Calc_RPM_Privod"
BEGIN
END_DATA_BLOCK

DATA_BLOCK "PaperVedVal2"	// DB 124
VERSION : 0.0
"Calc_RPM_Privod"
BEGIN
END_DATA_BLOCK

DATA_BLOCK "CalcRPM_PapVedVal3"	// DB 125
VERSION : 0.0
"Calc_RPM_Privod"
BEGIN
END_DATA_BLOCK

DATA_BLOCK "CalcRPM_RozgonTambur"	// DB 126
VERSION : 0.0
"Calc_RPM_Privod"
BEGIN
END_DATA_BLOCK

DATA_BLOCK "SpeedCalc_KombiPress"	// DB 130
VERSION : 0.0
"Calc_Speed_Unit"
BEGIN
END_DATA_BLOCK

DATA_BLOCK "SpeedCalc_Sitka"	// DB 131
VERSION : 0.0
"Calc_Speed_Unit"
BEGIN
END_DATA_BLOCK

DATA_BLOCK "CalcSpeed_Pres3"	// DB 132
VERSION : 0.0
"Calc_Speed_Unit"
BEGIN
END_DATA_BLOCK

DATA_BLOCK "CalcSpeed_Sushka1"	// DB 133
VERSION : 0.0
"Calc_Speed_Unit"
BEGIN
END_DATA_BLOCK

DATA_BLOCK "CalcSpeed_Sushka2"	// DB 134
VERSION : 0.0
"Calc_Speed_Unit"
BEGIN
END_DATA_BLOCK

DATA_BLOCK "CalcSpeed_Sushka3"	// DB 135
VERSION : 0.0
"Calc_Speed_Unit"
BEGIN
END_DATA_BLOCK

DATA_BLOCK "CalcSpeed_Sushka4"	// DB 136
VERSION : 0.0
"Calc_Speed_Unit"
BEGIN
END_DATA_BLOCK

DATA_BLOCK "CalcSpeed_KlejPress"	// DB 137
VERSION : 0.0
"Calc_Speed_Unit"
BEGIN
END_DATA_BLOCK

DATA_BLOCK "CalcSpeed_Sushka5"	// DB 138
VERSION : 0.0
"Calc_Speed_Unit"
BEGIN
END_DATA_BLOCK

DATA_BLOCK "CalcSpeed_Sushka6"	// DB 139
VERSION : 0.0
"Calc_Speed_Unit"
BEGIN
END_DATA_BLOCK

DATA_BLOCK "CalcSpeed_Sushka7"	// DB 140
VERSION : 0.0
"Calc_Speed_Unit"
BEGIN
END_DATA_BLOCK

DATA_BLOCK DB 141
VERSION : 0.0
"Calc_Speed_Unit"
BEGIN
END_DATA_BLOCK

DATA_BLOCK DB 142
VERSION : 0.0
"Calc_Speed_Unit"
BEGIN
END_DATA_BLOCK

DATA_BLOCK DB 200
VERSION : 0.1
  STRUCT
   Nakat_on : BOOL ;	//Pusk nakat z plc nakat
   rTambur_on : BOOL ;	//Pusk Rozg tambur z plc nakat
   bool_rezerv : ARRAY  [1 .. 62 ] OF BOOL ;
   Corect_Sp_Nakat : INT ;
   Corect_Sp_Rozg_Tamb : INT ;
   int_rezerv : ARRAY  [1 .. 20 ] OF INT ;
  END_STRUCT ;	
BEGIN
END_DATA_BLOCK

DATA_BLOCK "Signals_To_Nakat"	// DB 201
VERSION : 0.1
  STRUCT
   Got_kalandr : BOOL ;	//Gotovnist Kalandr
   Got_Rozg_Tambur : BOOL ;	//Gotovnist Rozgoni Tambur
   Got_Nakat : BOOL ;	//Gotovnist Rozgoni Nakat
   rezerv_bool : ARRAY  [1 .. 63 ] OF BOOL ;
   Speed_Suchka7_di : DINT ;
   Nakat_CurSpeed : WORD ;	//Current Speed Nakat
   RozgonTambur_CurSpeed : WORD ;	//CurrentSpeed Rozg Tambur
  END_STRUCT ;	
BEGIN
END_DATA_BLOCK

DATA_BLOCK DB 202
AUTHOR : SIMATIC
FAMILY : COM_FUNC
VERSION : 0.0
"GET"
BEGIN
END_DATA_BLOCK

DATA_BLOCK "PapVed1_Speed_Unit"	// DB 203
VERSION : 0.0
"Calc_Speed_Unit"
BEGIN
END_DATA_BLOCK

DATA_BLOCK "PapVed2_Speed_Unit"	// DB 204
VERSION : 0.0
"Calc_Speed_Unit"
BEGIN
END_DATA_BLOCK

DATA_BLOCK "PapVed3_Speed_Unit"	// DB 205
VERSION : 0.0
"Calc_Speed_Unit"
BEGIN
END_DATA_BLOCK

ORGANIZATION_BLOCK OB 1
TITLE = "Main Program Sweep (Cycle)"
VERSION : 0.1
VAR_TEMP
  OB1_EV_CLASS : BYTE ;	//Bits 0-3 = 1 (Coming event), Bits 4-7 = 1 (Event class 1)
  OB1_SCAN_1 : BYTE ;	//1 (Cold restart scan 1 of OB 1), 3 (Scan 2-n of OB 1)
  OB1_PRIORITY : BYTE ;	//Priority of OB Execution
  OB1_OB_NUMBR : BYTE ;	//1 (Organization block 1, OB1)
  OB1_RESERVED_1 : BYTE ;	//Reserved for system
  OB1_RESERVED_2 : BYTE ;	//Reserved for system
  OB1_PREV_CYCLE : INT ;	//Cycle time of previous OB1 scan (milliseconds)
  OB1_MIN_CYCLE : INT ;	//Minimum cycle time of OB1 (milliseconds)
  OB1_MAX_CYCLE : INT ;	//Maximum cycle time of OB1 (milliseconds)
  OB1_DATE_TIME : DATE_AND_TIME ;	//Date and time OB1 started
  S_MASH_DI : DINT ;
  S_MASH : BOOL ;
  bypass : BOOL ;
END_VAR
BEGIN
NETWORK
TITLE = Отримати дані з ПЛК_Накат
      A     M 10.1;
      =     L 25.0;
      BLD   103;
      BLD   9;
      =     L 30.0;
      CDB;
      OPN   DI 202;
      TAR2  LD 26;
      A     L 25.0;
      =     DIX 0.0;
      L     1;
      T     DIW 2;
      L     W#16#1002;
      T     DIW 8;
      L     14;
      T     DIW 10;
      L     200;
      T     DIW 12;
      L     P#DBX 0.0;
      T     DID 14;
      L     W#16#1002;
      T     DIW 48;
      L     14;
      T     DIW 50;
      L     200;
      T     DIW 52;
      L     P#DBX 0.0;
      T     DID 54;
      LAR2  P#DBX 0.0;
      UC    "GET";
      LAR2  LD 26;
      CDB;
      BLD   10;
      NOP   0;
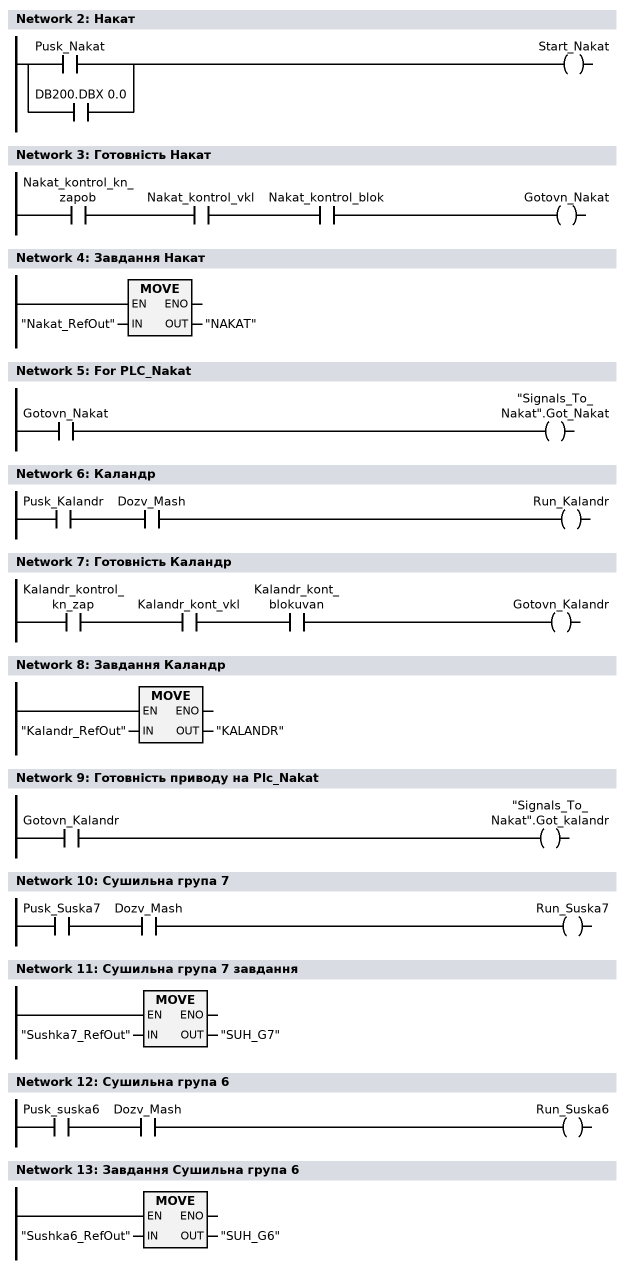
NETWORK
TITLE = Накат
//*******************
//Включити
//
      O     "Pusk_Nakat";
      O     DB200.DBX 0.0;
      =     "Start_Nakat";
NETWORK
TITLE = Готовність Накат
      A     "Nakat_kontrol_kn_zapob";
      A     "Nakat_kontrol_vkl";
      A     "Nakat_kontrol_blok";
      =     "Gotovn_Nakat";
NETWORK
TITLE = Завдання Накат
      L     "Nakat_RefOut";
      T     "NAKAT";
      NOP   0;
NETWORK
TITLE = For PLC_Nakat
      A     "Gotovn_Nakat";
      =     "Signals_To_Nakat".Got_Nakat;
NETWORK
TITLE = Каландр
//*********************
//Включити
//
      A     "Pusk_Kalandr";
      A     "Dozv_Mash";
      =     "Run_Kalandr";
NETWORK
TITLE = Готовність Каландр 
      A     "Kalandr_kontrol_kn_zap";
      A     "Kalandr_kont_vkl";
      A     "Kalandr_kont_blokuvan";
      =     "Gotovn_Kalandr";
NETWORK
TITLE = Завдання Каландр
      L     "Kalandr_RefOut";
      T     "KALANDR";
      NOP   0;
NETWORK
TITLE = Готовність приводу на Plc_Nakat
      A     "Gotovn_Kalandr";
      =     "Signals_To_Nakat".Got_kalandr;
NETWORK
TITLE = Сушильна група 7
//******************************
//
      A     "Pusk_Suska7";
      A     "Dozv_Mash";
      =     "Run_Suska7";
NETWORK
TITLE = Сушильна група 7 завдання
      L     "Sushka7_RefOut";
      T     "SUH_G7";
      NOP   0;
NETWORK
TITLE = Сушильна група 6
//******************************
//Включити
      A     "Pusk_suska6";
      A     "Dozv_Mash";
      =     "Run_Suska6";
NETWORK
TITLE = Завдання Сушильна група 6
      L     "Sushka6_RefOut";
      T     "SUH_G6";
      NOP   0;
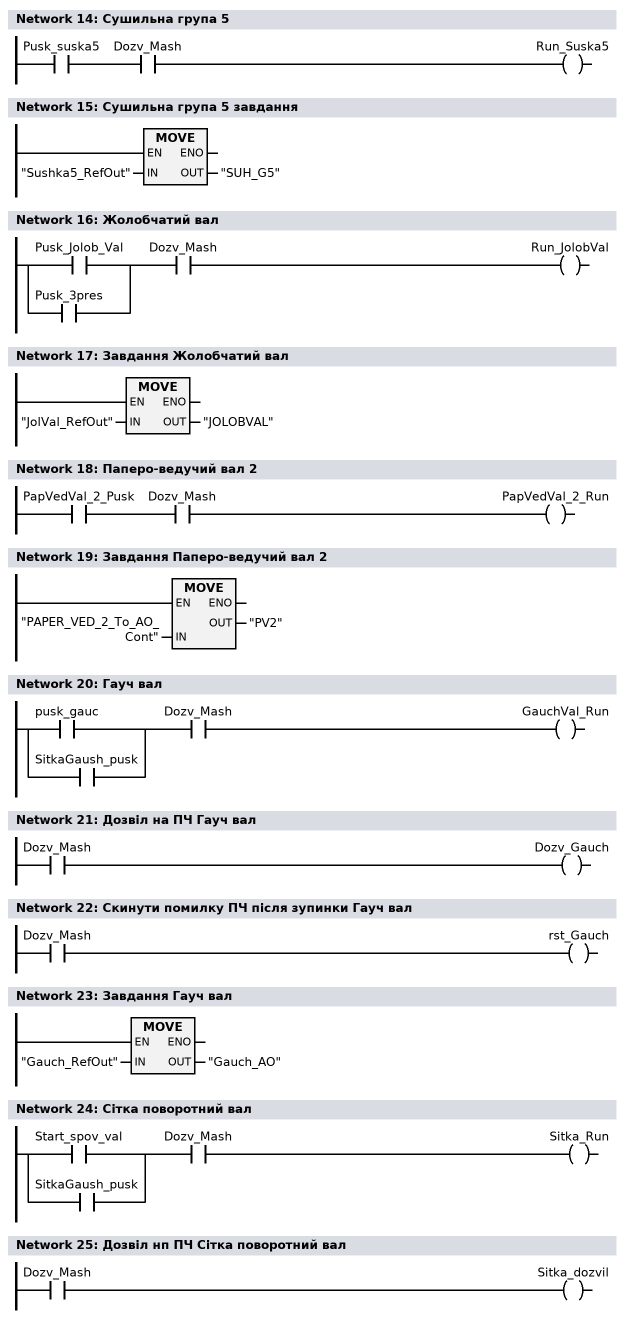
NETWORK
TITLE = Сушильна група 5 
//******************************
      A     "Pusk_suska5";
      A     "Dozv_Mash";
      =     "Run_Suska5";
NETWORK
TITLE = Сушильна група 5 завдання
      L     "Sushka5_RefOut";
      T     "SUH_G5";
      NOP   0;
NETWORK
TITLE = Жолобчатий вал
//****************************
//Включити
      A(;
      O     "Pusk_Jolob_Val";
      O     "Pusk_3pres";
      );
      A     "Dozv_Mash";
      =     "Run_JolobVal";
NETWORK
TITLE = Завдання Жолобчатий вал
      L     "JolVal_RefOut";
      T     "JOLOBVAL";
      NOP   0;
NETWORK
TITLE = Паперо-ведучий вал 2
//**********************************
//Включити
      A     "PapVedVal_2_Pusk";
      A     "Dozv_Mash";
      =     "PapVedVal_2_Run";
NETWORK
TITLE = Завдання Паперо-ведучий вал 2
      L     "PAPER_VED_2_To_AO_Cont";
      T     "PV2";
      NOP   0;
NETWORK
TITLE = Гауч вал
//**********************
//Включити
      A(;
      O     "pusk_gauc";
      O     "SitkaGaush_pusk";
      );
      A     "Dozv_Mash";
      =     "GauchVal_Run";
NETWORK
TITLE = Дозвіл на ПЧ Гауч вал
      A     "Dozv_Mash";
      =     "Dozv_Gauch";
NETWORK
TITLE = Скинути помилку ПЧ після зупинки Гауч вал
      A     "Dozv_Mash";
      =     "rst_Gauch";
NETWORK
TITLE = Завдання Гауч вал
      L     "Gauch_RefOut";
      T     "Gauch_AO";
      NOP   0;
NETWORK
TITLE = Сітка поворотний вал
//*********************************
//Включити
      A(;
      O     "Start_spov_val";
      O     "SitkaGaush_pusk";
      );
      A     "Dozv_Mash";
      =     "Sitka_Run";
NETWORK
TITLE = Дозвіл нп ПЧ Сітка поворотний вал
      A     "Dozv_Mash";
      =     "Sitka_dozvil";
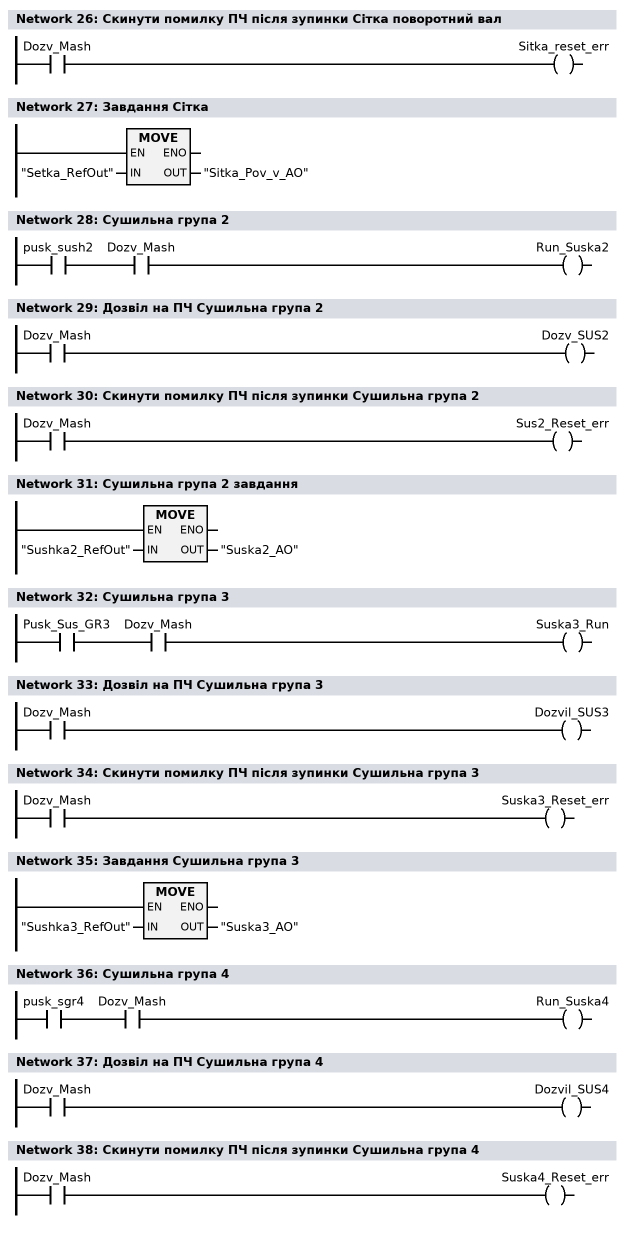
NETWORK
TITLE = Скинути помилку ПЧ після зупинки Сітка поворотний вал
      A     "Dozv_Mash";
      =     "Sitka_reset_err";
NETWORK
TITLE = Завдання Сітка
      L     "Setka_RefOut";
      T     "Sitka_Pov_v_AO";
      NOP   0;
NETWORK
TITLE = Сушильна група 2
//****************************
//Включити
      A     "pusk_sush2";
      A     "Dozv_Mash";
      =     "Run_Suska2";
NETWORK
TITLE = Дозвіл на ПЧ Сушильна група 2
      A     "Dozv_Mash";
      =     "Dozv_SUS2";
NETWORK
TITLE = Скинути помилку ПЧ після зупинки Сушильна група 2 
      A     "Dozv_Mash";
      =     "Sus2_Reset_err";
NETWORK
TITLE = Сушильна група 2 завдання
      L     "Sushka2_RefOut";
      T     "Suska2_AO";
      NOP   0;
NETWORK
TITLE = Сушильна група 3
//****************************
//Включити
      A     "Pusk_Sus_GR3";
      A     "Dozv_Mash";
      =     "Suska3_Run";
NETWORK
TITLE = Дозвіл на ПЧ Сушильна група 3
      A     "Dozv_Mash";
      =     "Dozvil_SUS3";
NETWORK
TITLE = Скинути помилку ПЧ після зупинки Сушильна група 3
      A     "Dozv_Mash";
      =     "Suska3_Reset_err";
NETWORK
TITLE = Завдання Сушильна група 3
      L     "Sushka3_RefOut";
      T     "Suska3_AO";
      NOP   0;
NETWORK
TITLE = Сушильна група 4
//****************************
//Включити
      A     "pusk_sgr4";
      A     "Dozv_Mash";
      =     "Run_Suska4";
NETWORK
TITLE = Дозвіл на ПЧ Сушильна група 4
      A     "Dozv_Mash";
      =     "Dozvil_SUS4";
NETWORK
TITLE = Скинути помилку ПЧ після зупинки Сушильна група 4
      A     "Dozv_Mash";
      =     "Suska4_Reset_err";
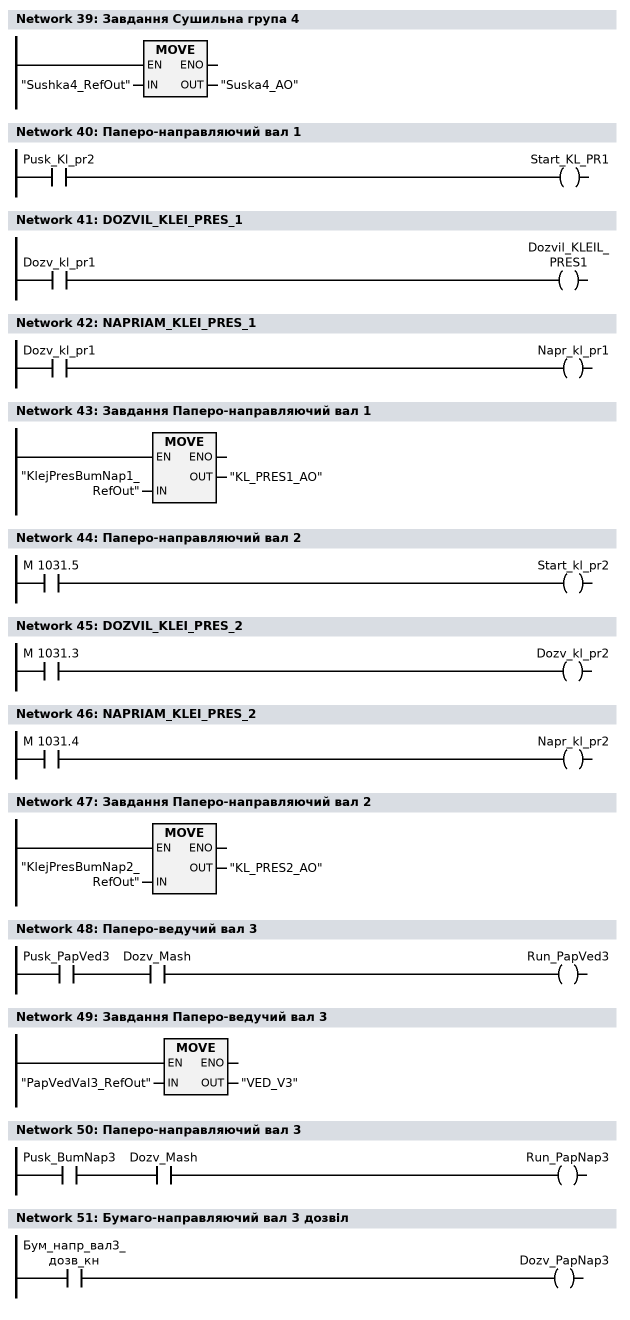
NETWORK
TITLE = Завдання Сушильна група 4
      L     "Sushka4_RefOut";
      T     "Suska4_AO";
      NOP   0;
NETWORK
TITLE = Паперо-направляючий вал 1
//                  ***Клей прес ***
//Включити
      A     "Pusk_Kl_pr2";
      =     "Start_KL_PR1";
NETWORK
TITLE = DOZVIL_KLEI_PRES_1
      A     "Dozv_kl_pr1";
      =     "Dozvil_KLEIL_PRES1";
NETWORK
TITLE = NAPRIAM_KLEI_PRES_1
      A     "Dozv_kl_pr1";
      =     "Napr_kl_pr1";
NETWORK
TITLE = Завдання Паперо-направляючий вал 1
      L     "KlejPresBumNap1_RefOut";
      T     "KL_PRES1_AO";
      NOP   0;
NETWORK
TITLE = Паперо-направляючий вал 2
//                  ***Клей прес***
//Включити
      A     M 1031.5;
      =     "Start_kl_pr2";
NETWORK
TITLE = DOZVIL_KLEI_PRES_2
      A     M 1031.3;
      =     "Dozv_kl_pr2";
NETWORK
TITLE = NAPRIAM_KLEI_PRES_2
      A     M 1031.4;
      =     "Napr_kl_pr2";
NETWORK
TITLE = Завдання Паперо-направляючий вал 2
      L     "KlejPresBumNap2_RefOut";
      T     "KL_PRES2_AO";
      NOP   0;
NETWORK
TITLE = Паперо-ведучий вал 3
//**********************************
//Включити
      A     "Pusk_PapVed3";
      A     "Dozv_Mash";
      =     "Run_PapVed3";
NETWORK
TITLE = Завдання Паперо-ведучий вал 3
      L     "PapVedVal3_RefOut";
      T     "VED_V3";
      NOP   0;
NETWORK
TITLE = Паперо-направляючий вал 3 
//****************************************
//Включити
      A     "Pusk_BumNap3";
      A     "Dozv_Mash";
      =     "Run_PapNap3";
NETWORK
TITLE = Бумаго-направляючий вал 3 дозвіл
      A     "Бум_напр_вал3_дозв_кн";
      =     "Dozv_PapNap3";
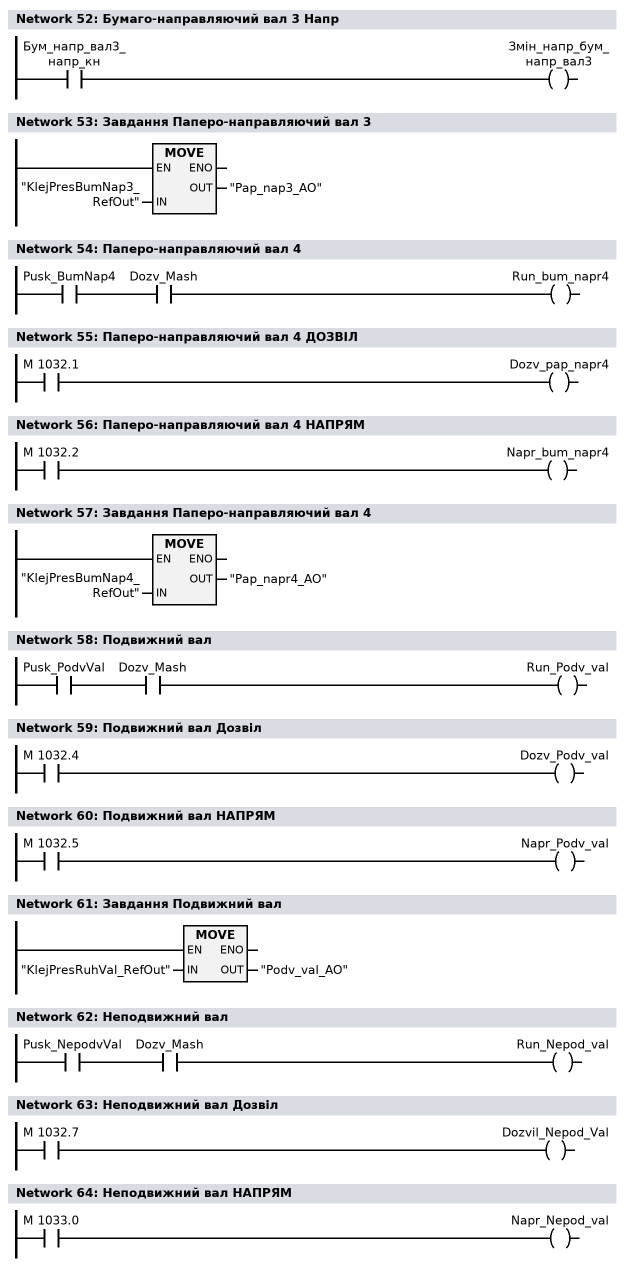
NETWORK
TITLE = Бумаго-направляючий вал 3 Напр
      A     "Бум_напр_вал3_напр_кн";
      =     "Змін_напр_бум_напр_вал3";
NETWORK
TITLE = Завдання Паперо-направляючий вал 3
      L     "KlejPresBumNap3_RefOut";
      T     "Pap_nap3_AO";
      NOP   0;
NETWORK
TITLE = Паперо-направляючий вал 4 
//                 ***Клей прес***
//Включити
      A     "Pusk_BumNap4";
      A     "Dozv_Mash";
      =     "Run_bum_napr4";
NETWORK
TITLE = Паперо-направляючий вал 4 ДОЗВІЛ
      A     M 1032.1;
      =     "Dozv_pap_napr4";
NETWORK
TITLE = Паперо-направляючий вал 4 НАПРЯМ
      A     M 1032.2;
      =     "Napr_bum_napr4";
NETWORK
TITLE = Завдання Паперо-направляючий вал 4
      L     "KlejPresBumNap4_RefOut";
      T     "Pap_napr4_AO";
      NOP   0;
NETWORK
TITLE = Подвижний вал 
//          ***Клей прес***
//Включити
      A     "Pusk_PodvVal";
      A     "Dozv_Mash";
      =     "Run_Podv_val";
NETWORK
TITLE = Подвижний вал Дозвіл
      A     M 1032.4;
      =     "Dozv_Podv_val";
NETWORK
TITLE = Подвижний вал НАПРЯМ
      A     M 1032.5;
      =     "Napr_Podv_val";
NETWORK
TITLE = Завдання Подвижний вал
      L     "KlejPresRuhVal_RefOut";
      T     "Podv_val_AO";
      NOP   0;
NETWORK
TITLE = Неподвижний вал 
//        ***Клей прес***
//Включити
      A     "Pusk_NepodvVal";
      A     "Dozv_Mash";
      =     "Run_Nepod_val";
NETWORK
TITLE = Неподвижний вал Дозвіл
      A     M 1032.7;
      =     "Dozvil_Nepod_Val";
NETWORK
TITLE = Неподвижний вал НАПРЯМ
      A     M 1033.0;
      =     "Napr_Nepod_val";
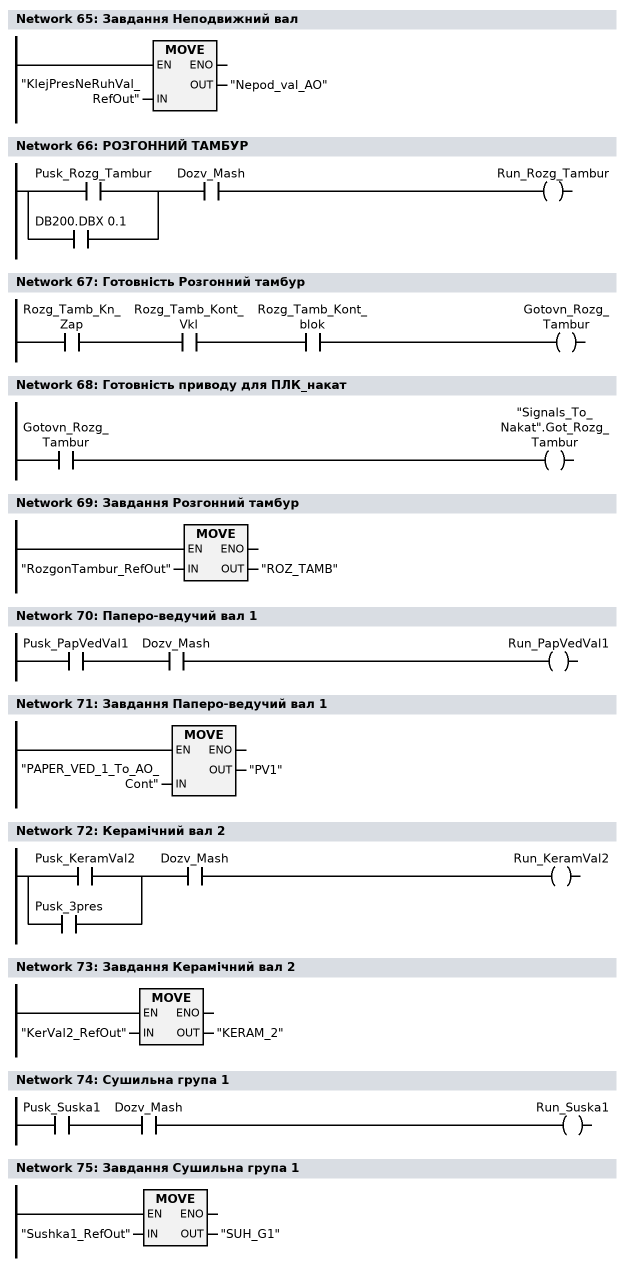
NETWORK
TITLE = Завдання Неподвижний вал
      L     "KlejPresNeRuhVal_RefOut";
      T     "Nepod_val_AO";
      NOP   0;
NETWORK
TITLE = РОЗГОННИЙ ТАМБУР
//******************************
//Включити
      A(;
      O     "Pusk_Rozg_Tambur";
      O     DB200.DBX 0.1;
      );
      A     "Dozv_Mash";
      =     "Run_Rozg_Tambur";
NETWORK
TITLE = Готовність Розгонний тамбур
      A     "Rozg_Tamb_Kn_Zap";
      A     "Rozg_Tamb_Kont_Vkl";
      A     "Rozg_Tamb_Kont_blok";
      =     "Gotovn_Rozg_Tambur";
NETWORK
TITLE = Готовність приводу для ПЛК_накат
      A     "Gotovn_Rozg_Tambur";
      =     "Signals_To_Nakat".Got_Rozg_Tambur;
NETWORK
TITLE = Завдання Розгонний тамбур
      L     "RozgonTambur_RefOut";
      T     "ROZ_TAMB";
      NOP   0;
NETWORK
TITLE = Паперо-ведучий вал 1
//*************************
//Включити
      A     "Pusk_PapVedVal1";
      A     "Dozv_Mash";
      =     "Run_PapVedVal1";
NETWORK
TITLE = Завдання Паперо-ведучий вал 1
      L     "PAPER_VED_1_To_AO_Cont";
      T     "PV1";
      NOP   0;
NETWORK
TITLE = Керамічний вал 2
//******************************
//Включити
      A(;
      O     "Pusk_KeramVal2";
      O     "Pusk_3pres";
      );
      A     "Dozv_Mash";
      =     "Run_KeramVal2";
NETWORK
TITLE = Завдання Керамічний вал 2
      L     "KerVal2_RefOut";
      T     "KERAM_2";
      NOP   0;
NETWORK
TITLE = Сушильна група 1
//*************************
//Включити
      A     "Pusk_Suska1";
      A     "Dozv_Mash";
      =     "Run_Suska1";
NETWORK
TITLE = Завдання Сушильна група 1
      L     "Sushka1_RefOut";
      T     "SUH_G1";
      NOP   0;
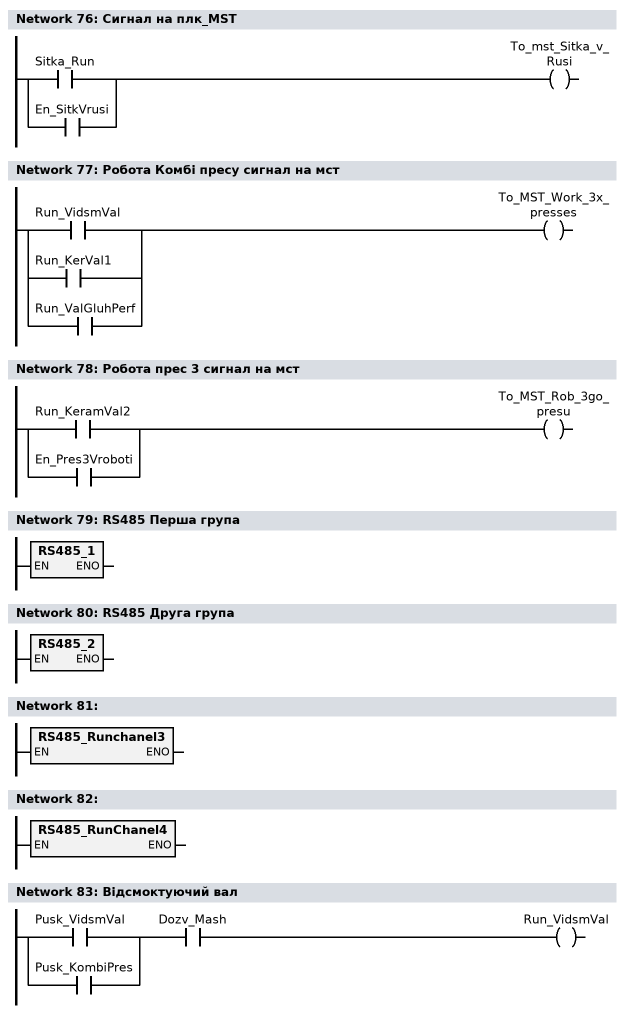
NETWORK
TITLE = Сигнал на плк_MST 
//                   ***MST***
//Сітка в роботі
      O     "Sitka_Run";
      O     "En_SitkVrusi";
      =     "To_mst_Sitka_v_Rusi";
NETWORK
TITLE = Робота Комбі пресу сигнал на мст
      O     "Run_VidsmVal";
      O     "Run_KerVal1";
      O     "Run_ValGluhPerf";
      =     "To_MST_Work_3x_presses";
NETWORK
TITLE = Робота прес 3 сигнал на мст
      O     "Run_KeramVal2";
      O     "En_Pres3Vroboti";
      =     "To_MST_Rob_3go_presu";
NETWORK
TITLE = RS485 Перша група
      CALL  "RS485_1";
      NOP   0;
NETWORK
TITLE = RS485 Друга група
      CALL  "RS485_2";
      NOP   0;
NETWORK
TITLE =
      CALL  "RS485_Runchanel3";
      NOP   0;
NETWORK
TITLE =
      CALL  "RS485_RunChanel4";
      NOP   0;
NETWORK
TITLE = Відсмоктуючий вал
//***********************************
//Включити
      A(;
      O     "Pusk_VidsmVal";
      O     "Pusk_KombiPres";
      );
      A     "Dozv_Mash";
      =     "Run_VidsmVal";
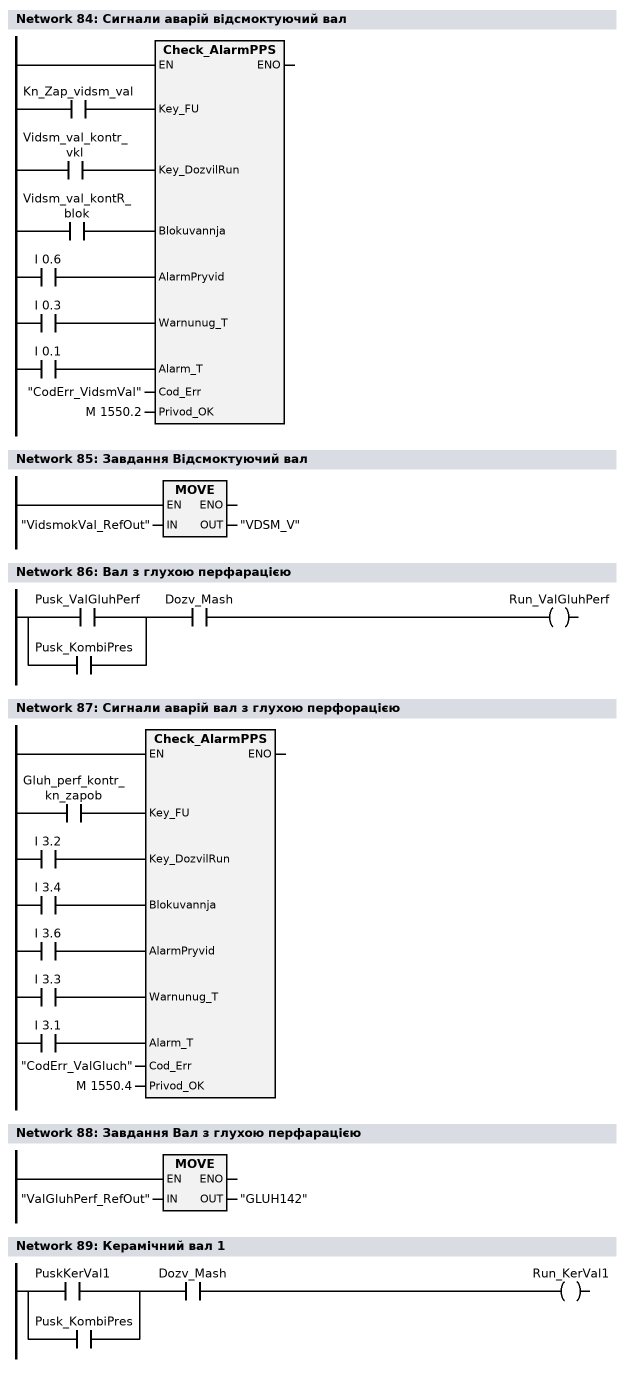
NETWORK
TITLE = Сигнали аварій відсмоктуючий вал
      A     "Kn_Zap_vidsm_val";
      =     L 25.0;
      BLD   103;
      A     "Vidsm_val_kontr_vkl";
      =     L 25.1;
      BLD   103;
      A     "Vidsm_val_kontR_blok";
      =     L 25.2;
      BLD   103;
      A     I 0.6;
      =     L 25.3;
      BLD   103;
      A     I 0.3;
      =     L 25.4;
      BLD   103;
      A     I 0.1;
      =     L 25.5;
      BLD   103;
      CALL  "Check_AlarmPPS" (
           Key_FU                   := L 25.0,
           Key_DozvilRun            := L 25.1,
           Blokuvannja              := L 25.2,
           AlarmPryvid              := L 25.3,
           Warnunug_T               := L 25.4,
           Alarm_T                  := L 25.5,
           Cod_Err                  := "CodErr_VidsmVal",
           Privod_OK                := M 1550.2);
      NOP   0;
NETWORK
TITLE = Завдання Відсмоктуючий вал
      L     "VidsmokVal_RefOut";
      T     "VDSM_V";
      NOP   0;
NETWORK
TITLE = Вал з глухою перфарацією
//*********************************************
//Включити
      A(;
      O     "Pusk_ValGluhPerf";
      O     "Pusk_KombiPres";
      );
      A     "Dozv_Mash";
      =     "Run_ValGluhPerf";
NETWORK
TITLE = Сигнали аварій вал з глухою перфорацією
      A     "Gluh_perf_kontr_kn_zapob";
      =     L 25.0;
      BLD   103;
      A     I 3.2;
      =     L 25.1;
      BLD   103;
      A     I 3.4;
      =     L 25.2;
      BLD   103;
      A     I 3.6;
      =     L 25.3;
      BLD   103;
      A     I 3.3;
      =     L 25.4;
      BLD   103;
      A     I 3.1;
      =     L 25.5;
      BLD   103;
      CALL  "Check_AlarmPPS" (
           Key_FU                   := L 25.0,
           Key_DozvilRun            := L 25.1,
           Blokuvannja              := L 25.2,
           AlarmPryvid              := L 25.3,
           Warnunug_T               := L 25.4,
           Alarm_T                  := L 25.5,
           Cod_Err                  := "CodErr_ValGluch",
           Privod_OK                := M 1550.4);
      NOP   0;
NETWORK
TITLE = Завдання Вал з глухою перфарацією
      L     "ValGluhPerf_RefOut";
      T     "GLUH142";
      NOP   0;
NETWORK
TITLE = Керамічний вал 1
//****************************************
//Включити
      A(;
      O     "PuskKerVal1";
      O     "Pusk_KombiPres";
      );
      A     "Dozv_Mash";
      =     "Run_KerVal1";
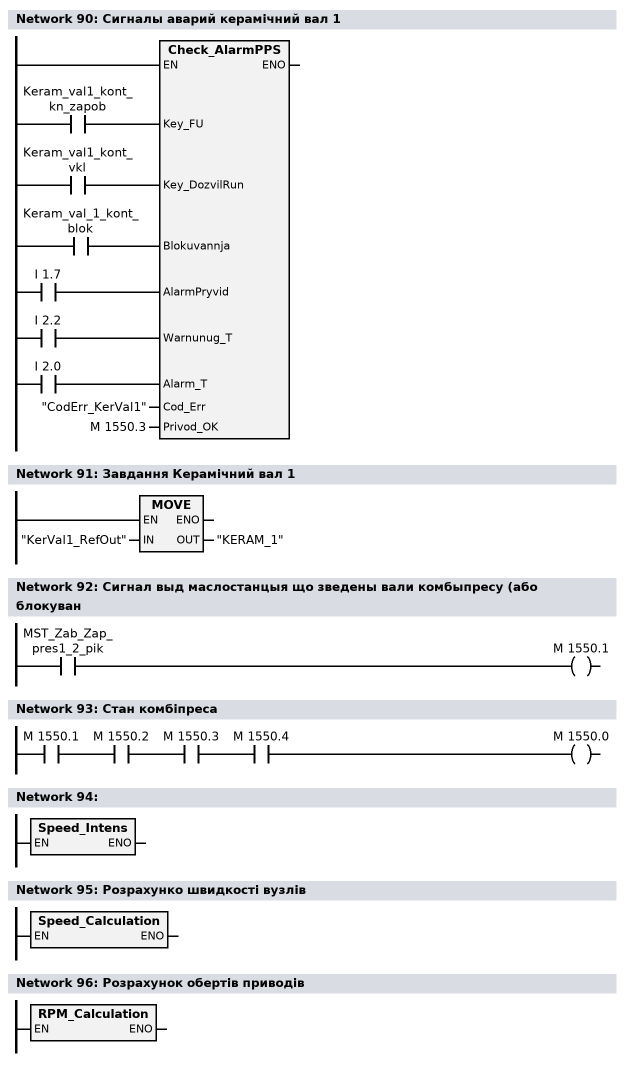
NETWORK
TITLE = Сигналы аварий керамічний вал 1
      A     "Keram_val1_kont_kn_zapob";
      =     L 25.0;
      BLD   103;
      A     "Keram_val1_kont_vkl";
      =     L 25.1;
      BLD   103;
      A     "Keram_val_1_kont_blok";
      =     L 25.2;
      BLD   103;
      A     I 1.7;
      =     L 25.3;
      BLD   103;
      A     I 2.2;
      =     L 25.4;
      BLD   103;
      A     I 2.0;
      =     L 25.5;
      BLD   103;
      CALL  "Check_AlarmPPS" (
           Key_FU                   := L 25.0,
           Key_DozvilRun            := L 25.1,
           Blokuvannja              := L 25.2,
           AlarmPryvid              := L 25.3,
           Warnunug_T               := L 25.4,
           Alarm_T                  := L 25.5,
           Cod_Err                  := "CodErr_KerVal1",
           Privod_OK                := M 1550.3);
      NOP   0;
NETWORK
TITLE = Завдання Керамічний вал 1
      L     "KerVal1_RefOut";
      T     "KERAM_1";
      NOP   0;
NETWORK
TITLE = Сигнал выд маслостанцыя що зведены вали комбыпресу (або блокуван
      A     "MST_Zab_Zap_pres1_2_pik";
      =     M 1550.1;
NETWORK
TITLE = Стан комбіпреса
      A     M 1550.1;
      A     M 1550.2;
      A     M 1550.3;
      A     M 1550.4;
      =     M 1550.0;
NETWORK
TITLE =
      CALL  "Speed_Intens";
      NOP   0;
NETWORK
TITLE = Розрахунко швидкості вузлів
      CALL  "Speed_Calculation";
      NOP   0;
NETWORK
TITLE = Розрахунок обертів приводів
      CALL  "RPM_Calculation";
      NOP   0;
END_ORGANIZATION_BLOCK

ORGANIZATION_BLOCK "COMPLETE RESTART"	// OB 100
TITLE = "Complete Restart"
VERSION : 0.1
VAR_TEMP
  OB100_EV_CLASS : BYTE ;	//16#13, Event class 1, Entering event state, Event logged in diagnostic buffer
  OB100_STRTUP : BYTE ;	//16#81/82/83/84 Method of startup
  OB100_PRIORITY : BYTE ;	//Priority of OB Execution
  OB100_OB_NUMBR : BYTE ;	//100 (Organization block 100, OB100)
  OB100_RESERVED_1 : BYTE ;	//Reserved for system
  OB100_RESERVED_2 : BYTE ;	//Reserved for system
  OB100_STOP : WORD ;	//Event that caused CPU to stop (16#4xxx)
  OB100_STRT_INFO : DWORD ;	//Information on how system started
  OB100_DATE_TIME : DATE_AND_TIME ;	//Date and time OB100 started
END_VAR
BEGIN
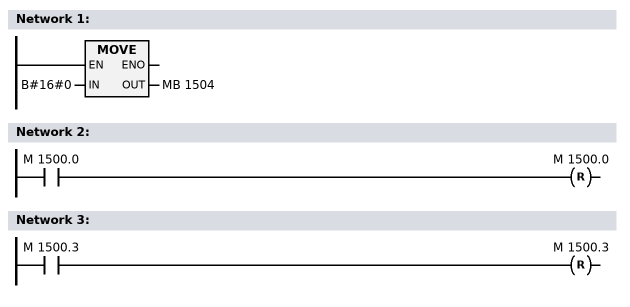
NETWORK
TITLE =
      L     B#16#0;
      T     MB 1504;
      NOP   0;
NETWORK
TITLE =
      A     M 1500.0;
      R     M 1500.0;
NETWORK
TITLE =
      A     M 1500.3;
      R     M 1500.3;
END_ORGANIZATION_BLOCK
